// TwinCAT 3 PLC project Untitled1
// ProgramVersion: 3.1.4024.0
// libraries:
//   Tc2_EtherCAT, * (Beckhoff Automation GmbH)
//   Tc2_MC2, * (Beckhoff Automation GmbH)
//   Tc2_ModbusSrv, * (Beckhoff Automation GmbH)
//   Tc2_Standard, * (Beckhoff Automation GmbH)
//   Tc2_SUPS, * (Beckhoff Automation GmbH)
//   Tc2_System, * (Beckhoff Automation GmbH)
//   Tc2_Utilities, * (Beckhoff Automation GmbH)
//   Tc3_Module, * (Beckhoff Automation GmbH)
//   Util, * (System)
//   VisuDialogs, * (System)
// project tree:
//   02DUTs/Ads/ AutostoreControlCommand.TcDUT (not stored), AutostoreStatus.TcDUT, BarcodeVerificationResult.TcDUT, ButtonStatus.TcDUT, DigitalInputStatus.TcDUT (not stored), DigitalOutputStatus.TcDUT (not stored), EStopStatus.TcDUT, E_SAFETYDOOR.TcDUT, E_SafetyStates.TcDUT, FB_Application.TcPOU, FB_Light_tower_module.TcPOU, FB_Safety_module.TcPOU, FB_ToteData.TcPOU, FB_Tote_Subsystem.TcPOU, MachineControlCommand.TcDUT, MachineStatus.TcDUT, OrderToteCommand.TcDUT, OrderToteErrorStatus.TcDUT, SafetyDoorStatus.TcDUT, SafetyStatus.TcDUT, StationMode.TcDUT, ST_IO_16.TcDUT (not stored), ST_LightTower.TcDUT, ToteStatus.TcDUT, ToteSubsystemWorkflowStatus.TcDUT
//   GVLs/ GVL.TcGVL, GVL_IOLink.TcGVL, G_HMI.TcGVL, G_IO.TcGVL
//   / EtherCAT_Task.TcTTO, GlobalTextList.TcGTLO, MianTask.TcTTO, VisualizationManager.TcVMO (not stored), VISU_TASK.TcTTO
//   Mian/ Event_add.TcPOU, Event_clear.TcPOU, MAIN.TcPOU
//   Mian/machine/axis/ AxisHMI_Ex.TcVIS (not stored), E_HomingSteps.TcDUT (not stored), FB_MotionAxis_MC.TcPOU, MC_HomeAxis.TcPOU (not stored), ST_MotionAxis_MC.TcDUT
//   Mian/machine/bufferr module/ Buffer_roller.TcDUT (not stored), E_RollerStates.TcDUT, FB_buffer.TcPOU, FB_roller.TcPOU, Inbound_roller.TcDUT
//   Mian/machine/ FB_DigitalInput.TcPOU (not stored), FB_GPWM.TcPOU (not stored), Roller.TcDUT, Valve.TcDUT (not stored)
//   Mian/machine/loading moudle/ E_LoadingStates.TcDUT, E_Transfer.TcDUT, FB_loading.TcPOU, Roller_x.TcDUT, Roller_y.TcDUT
//   Mian/machine/mcp/ FB_mcp.TcPOU, ST_control_pannel.TcDUT (not stored), ST_safetyDoor.TcDUT
//   Mian/machine/working moudle/Estates/ E_Condition.TcDUT, E_WorkingStates.TcDUT
//   Mian/machine/working moudle/ FB_working.TcPOU, Inbound.TcDUT, Outbound.TcDUT
//   Mian/statemachine/ E_SystemManager.TcDUT, Prepare_Date_Time.TcPOU, ST_EVENT.TcDUT (not stored)
//   VISUs/VISUs/ Menu.TcVIS, visu_buffer.TcVIS, visu_loading.TcVIS, visu_main.TcVIS, visu_operation.TcVIS, visu_working.TcVIS, v_io_buffer.TcVIS, v_alarm.TcVIS, v_io_loading.TcVIS, v_io_working.TcVIS
// real-time tasks:
//   TASK PlcTask: cycle T#10ms, priority 20, ADS port 350
//   TASK EtherCAT_Task: cycle T#2ms, priority 1, ADS port 351
//   TASK VISU_TASK: cycle T#200000us, priority 30, ADS port 352
// motion (NC):
//   TASK NC-Task 1 SAF: cycle T#4ms, priority 4, ADS port 501
//   TASK NC-Task 1 SVB: cycle T#10ms, priority 8, ADS port 511
//   AXIS buffer_stopper (id 1)
//     PositionAreaControl: Enable=false
//     OtherSettings: AllowMotionCmdToSlave=true
//     encoder EncType=19
//       EncPara: ScaleFactorNumerator=36, ScaleFactorDenominator=8388608, MaxCount=#xffffffff, ReferenceSystem=1
//         Inc: RefSoftSyncMask=#x00800000
//     drive DrvType=16
//       DrvPara: MaxCount=#xffffffff, DriveControlDWord=#x00020100
//         Analog: TorqueSetpointScale=10, ScaleFactorActTorque=0.1
//         TimeComp: TaskDelayCycles=1
//     controller CtrType=1
//       CtrPara: PriorControlFactor=1
//         PosDiffControl: Enable=false
//         Observer: BandWidth=20
//   AXIS lift_motor (id 3)
//     PositionAreaControl: Enable=false
//     OtherSettings: AllowMotionCmdToSlave=true
//     encoder EncType=19
//       EncPara: ScaleFactorNumerator=3.97364299e-07, MaxCount=#xffffffff, ReferenceSystem=1
//     drive DrvType=16
//       DrvPara: MaxCount=#xffffffff, DriveControlDWord=#x00020100
//         Analog: TorqueSetpointScale=10, ScaleFactorActTorque=0.1
//         TimeComp: TaskDelayCycles=1
//     controller CtrType=1
//       CtrPara: PriorControlFactor=1
//         PosDiffControl: Enable=false
//         Observer: BandWidth=20
//   AXIS working_lift_motor (id 4)
//     PositionAreaControl: Enable=false
//     OtherSettings: AllowMotionCmdToSlave=true
//     encoder EncType=19
//       EncPara: ScaleFactorNumerator=5.96046448e-07, Inverse=true, MaxCount=#xffffffff, ReferenceSystem=1
//     drive DrvType=16
//       DrvPara: Inverse=true, MaxCount=#xffffffff, DriveControlDWord=#x00020100
//         Analog: TorqueSetpointScale=10, ScaleFactorActTorque=0.1
//         TimeComp: TaskDelayCycles=1
//     controller CtrType=1
//       CtrPara: PriorControlFactor=1
//         PosDiffControl: Enable=false
//         Observer: BandWidth=20
//   AXIS working_open_bag (id 5)
//     General: UnitName=°
//     PositionAreaControl: Enable=false
//     OtherSettings: AllowMotionCmdToSlave=true
//     encoder EncType=1
//       EncPara: ScaleFactorNumerator=36, ScaleFactorDenominator=8388608, ReferenceSystem=1
//         Inc: RefSoftSyncMask=#x00800000
//     drive DrvType=5
//       Analog: TorqueSetpointScale=10, ScaleFactorActTorque=0.1
//       TimeComp: TaskDelayCycles=1
//     controller CtrType=1
//       CtrPara: PriorControlFactor=1
//         PosDiffControl: Enable=false
//         Observer: BandWidth=20
//   AXIS bag_open_vacuun_0 (id 2)
//     General: UnitName=°
//     PositionAreaControl: Enable=false
//     OtherSettings: AllowMotionCmdToSlave=true
//     encoder EncType=19
//       EncPara: ScaleFactorNumerator=90, ScaleFactorDenominator=8388608, MaxCount=#xffffffff, ReferenceSystem=1
//         Inc: RefSoftSyncMask=#x00800000
//     drive DrvType=16
//       DrvPara: MaxCount=#xffffffff, DriveControlDWord=#x00020100
//         Analog: TorqueSetpointScale=10, ScaleFactorActTorque=0.1
//         TimeComp: TaskDelayCycles=1
//     controller CtrType=1
//       CtrPara: PriorControlFactor=1
//         PosDiffControl: Enable=false
//         Observer: BandWidth=20
//   AXIS bag_open_vacuun_1 (id 8)
//     General: UnitName=°
//     PositionAreaControl: Enable=false
//     OtherSettings: AllowMotionCmdToSlave=true
//     encoder EncType=19
//       EncPara: ScaleFactorNumerator=90, ScaleFactorDenominator=8388608, MaxCount=#xffffffff, ReferenceSystem=1
//         Inc: RefSoftSyncMask=#x00800000
//     drive DrvType=16
//       DrvPara: MaxCount=#xffffffff, DriveControlDWord=#x00020100
//         Analog: TorqueSetpointScale=10, ScaleFactorActTorque=0.1
//         TimeComp: TaskDelayCycles=1
//     controller CtrType=1
//       CtrPara: PriorControlFactor=1
//         PosDiffControl: Enable=false
//         Observer: BandWidth=20
//   AXIS bag_open_0 (id 9)
//     General: UnitName=°
//     PositionAreaControl: Enable=false
//     OtherSettings: AllowMotionCmdToSlave=true
//     encoder EncType=19
//       EncPara: ScaleFactorNumerator=360, ScaleFactorDenominator=8388608, MaxCount=#xffffffff, ReferenceSystem=1
//         Inc: RefSoftSyncMask=#x00800000
//     drive DrvType=16
//       DrvPara: MaxCount=#xffffffff, DriveControlDWord=#x00020100
//         Analog: TorqueSetpointScale=10, ScaleFactorActTorque=0.1
//         TimeComp: TaskDelayCycles=1
//     controller CtrType=1
//       CtrPara: PriorControlFactor=1
//         PosDiffControl: Enable=false
//         Observer: BandWidth=20
//   AXIS bag_open_1 (id 7)
//     General: UnitName=°
//     PositionAreaControl: Enable=false
//     OtherSettings: AllowMotionCmdToSlave=true
//     encoder EncType=19
//       EncPara: ScaleFactorNumerator=360, ScaleFactorDenominator=8388608, MaxCount=#xffffffff, ReferenceSystem=1
//         Inc: RefSoftSyncMask=#x00800000
//     drive DrvType=16
//       DrvPara: MaxCount=#xffffffff, DriveControlDWord=#x00020100
//         Analog: TorqueSetpointScale=10, ScaleFactorActTorque=0.1
//         TimeComp: TaskDelayCycles=1
//     controller CtrType=1
//       CtrPara: PriorControlFactor=1
//         PosDiffControl: Enable=false
//         Observer: BandWidth=20
//   AXIS bag_open_2 (id 10)
//     General: UnitName=°
//     PositionAreaControl: Enable=false
//     OtherSettings: AllowMotionCmdToSlave=true
//     encoder EncType=19
//       EncPara: ScaleFactorNumerator=360, ScaleFactorDenominator=8388608, MaxCount=#xffffffff, ReferenceSystem=1
//         Inc: RefSoftSyncMask=#x00800000
//     drive DrvType=16
//       DrvPara: MaxCount=#xffffffff, DriveControlDWord=#x00020100
//         Analog: TorqueSetpointScale=10, ScaleFactorActTorque=0.1
//         TimeComp: TaskDelayCycles=1
//     controller CtrType=1
//       CtrPara: PriorControlFactor=1
//         PosDiffControl: Enable=false
//         Observer: BandWidth=20
//   AXIS bag_open_3 (id 6)
//     General: UnitName=°
//     PositionAreaControl: Enable=false
//     OtherSettings: AllowMotionCmdToSlave=true
//     encoder EncType=19
//       EncPara: ScaleFactorNumerator=360, ScaleFactorDenominator=8388608, MaxCount=#xffffffff, ReferenceSystem=1
//         Inc: RefSoftSyncMask=#x00800000
//     drive DrvType=16
//       DrvPara: MaxCount=#xffffffff, DriveControlDWord=#x00020100
//         Analog: TorqueSetpointScale=10, ScaleFactorActTorque=0.1
//         TimeComp: TaskDelayCycles=1
//     controller CtrType=1
//       CtrPara: PriorControlFactor=1
//         PosDiffControl: Enable=false
//         Observer: BandWidth=20
// I/O:
//   DEVICE Device 1 (EtherCAT), AmsNetId 192.168.11.159.2.1
//     Term 1 (EK1200) [EK1200-5000 EtherCAT Power supply (2A E-Bus)]
//       mcp_di0 [EL1809 16Ch. Dig. Input 24V, 3ms]
//       mcp_do0 [EL2809-0015 16Ch. Dig. Output 24V DC, 0.35A, not short-circuit proof]
//       Term 4 (EL6910) [EL6910, TwinSAFE PLC]
//       Term 5 (EL1904) [EL1904, 4 Ch. Safety Input 24V, TwinSAFE]
//         modules: Module 1 (FSOES)
//       Term 6 (EL2904) [EL2904, 4 Ch. Safety Output 24V, 0.5A, TwinSAFE]
//         modules: Module 1 (FSOES), Module 2 (DO)
//       Term 41 (EL3064) [EL3064 4Ch. Ana. Input 0-10V]
//       Term 42 (EL6631-0010) [EL6631-0010 PROFINET IO Device]
//       Term 7 (EL9011) [EL9011 End Terminal]
//   DEVICE Device 4 (EtherCAT), AmsNetId 192.168.11.159.5.1
//     Box 8 (CU1128) [CU1128 6x EtherCAT junction]
//       buffer_io [EK1100 EtherCAT Coupler (2A E-Bus)]
//         buffer_di1 [EL1809 16Ch. Dig. Input 24V, 3ms]
//         buffer_di2 [EL1809 16Ch. Dig. Input 24V, 3ms]
//         buffer_do1 [EL2809-0015 16Ch. Dig. Output 24V DC, 0.35A, not short-circuit proof]
//         buffer_do2 [EL2809-0015 16Ch. Dig. Output 24V DC, 0.35A, not short-circuit proof] (disabled)
//         Term 14 (EL1904) [EL1904, 4 Ch. Safety Input 24V, TwinSAFE]
//           modules: Module 1 (FSOES)
//         Term 15 (EL2904) [EL2904, 4 Ch. Safety Output 24V, 0.5A, TwinSAFE]
//           modules: Module 1 (FSOES), Module 2 (DO)
//         Term 31 (EL9011) [EL9011 End Terminal]
//       buffer_stopper [SV660_1Axis_00915]
//       loading_io [EK1100 EtherCAT Coupler (2A E-Bus)]
//         lift_di3 [EL1809 16Ch. Dig. Input 24V, 3ms]
//         lift_di4 [EL1809 16Ch. Dig. Input 24V, 3ms]
//         lift_do3 [EL2809-0015 16Ch. Dig. Output 24V DC, 0.35A, not short-circuit proof]
//         lift_do4 [EL2809-0015 16Ch. Dig. Output 24V DC, 0.35A, not short-circuit proof]
//         Term 23 (EL1904) [EL1904, 4 Ch. Safety Input 24V, TwinSAFE]
//           modules: Module 1 (FSOES)
//         Term 24 (EL1904) [EL1904, 4 Ch. Safety Input 24V, TwinSAFE]
//           modules: Module 1 (FSOES)
//         Term 25 (EL2904) [EL2904, 4 Ch. Safety Output 24V, 0.5A, TwinSAFE]
//           modules: Module 1 (FSOES), Module 2 (DO)
//         Term 32 (EL9011) [EL9011 End Terminal]
//       loading_motor [SV635_1Axis_03411]
//       working_module [CU1128 6x EtherCAT junction - Dev A]
//         working_io [EK1100 EtherCAT Coupler (2A E-Bus)]
//           working_di5 [EL1809 16Ch. Dig. Input 24V, 3ms]
//           working_di6 [EL1809 16Ch. Dig. Input 24V, 3ms]
//           working_do5 [EL2809-0015 16Ch. Dig. Output 24V DC, 0.35A, not short-circuit proof]
//           working_do6 [EL2809-0015 16Ch. Dig. Output 24V DC, 0.35A, not short-circuit proof]
//           Term 33 (EL1904) [EL1904, 4 Ch. Safety Input 24V, TwinSAFE]
//             modules: Module 1 (FSOES)
//           Term 34 (EL2904) [EL2904, 4 Ch. Safety Output 24V, 0.5A, TwinSAFE]
//             modules: Module 1 (FSOES), Module 2 (DO)
//           Term 33 (EL9011) [EL9011 End Terminal]
//         working_liftmotor [SV635_1Axis_03411]
//         woking_openbag [SV635_1Axis_03411]
//         bag_open_dio [EK1100 EtherCAT Coupler (2A E-Bus)]
//           di7 [EL1809 16Ch. Dig. Input 24V, 3ms]
//           di8 [EL1809 16Ch. Dig. Input 24V, 3ms]
//           do7 [EL2809-0015 16Ch. Dig. Output 24V DC, 0.35A, not short-circuit proof]
//           Term 71 (EL9011) [EL9011 End Terminal]
//         bag_vacuun [SV660ND_2Axis_V1.00]
//           modules: Module 1 (CSP/CSV), Module 2 (CSP/CSV)
//         bag_open_0_1 [SV660ND_2Axis_V1.00]
//           modules: Module 1 (CSP/CSV), Module 2 (CSP/CSV)
//         bag_open_2_3 [SV660ND_2Axis_V1.00]
//           modules: Module 1 (CSP/CSV), Module 2 (CSP/CSV)
//       Term 37 (CU1128-C) [CU1128 6x EtherCAT junction - Dev B]
// variable links:
//   Device 1 (EtherCAT) <-> Device 1 (EtherCAT)/Term 1 (EK1200)/Term 4 (EL6910)
//     Term 1 (EK1200)/Term 5 (EL1904)/Module 1 (FSOES)/RxPDO/FSOE <-> ConnectionInputs/Message_3 TxPDO
//     Term 1 (EK1200)/Term 5 (EL1904)/Module 1 (FSOES)/TxPDO/FSOE <-> ConnectionOutputs/Message_3 RxPDO
//   Device 1 (EtherCAT) <-> Device 1 (EtherCAT)/Term 1 (EK1200)/Term 6 (EL2904)
//     Term 1 (EK1200)/Term 4 (EL6910)/ConnectionInputs/Message_4 TxPDO <-> Module 1 (FSOES)/RxPDO/FSOE
//     Term 1 (EK1200)/Term 4 (EL6910)/ConnectionOutputs/Message_4 RxPDO <-> Module 1 (FSOES)/TxPDO/FSOE
//   Device 1 (EtherCAT) <-> Device 4 (EtherCAT)/Box 8 (CU1128)/buffer_io/Term 14 (EL1904)
//     Term 1 (EK1200)/Term 4 (EL6910)/ConnectionInputs/Message_5 TxPDO <-> Module 1 (FSOES)/RxPDO/FSOE
//     Term 1 (EK1200)/Term 4 (EL6910)/ConnectionOutputs/Message_5 RxPDO <-> Module 1 (FSOES)/TxPDO/FSOE
//   Device 1 (EtherCAT) <-> Device 4 (EtherCAT)/Box 8 (CU1128)/buffer_io/Term 15 (EL2904)
//     Term 1 (EK1200)/Term 4 (EL6910)/ConnectionInputs/Message_6 TxPDO <-> Module 1 (FSOES)/RxPDO/FSOE
//     Term 1 (EK1200)/Term 4 (EL6910)/ConnectionOutputs/Message_6 RxPDO <-> Module 1 (FSOES)/TxPDO/FSOE
//   Device 1 (EtherCAT) <-> Device 4 (EtherCAT)/Box 8 (CU1128)/loading_io/Term 23 (EL1904)
//     Term 1 (EK1200)/Term 4 (EL6910)/ConnectionOutputs/Message_7 RxPDO <-> Module 1 (FSOES)/TxPDO/FSOE
//   Device 1 (EtherCAT) <-> Device 4 (EtherCAT)/Box 8 (CU1128)/loading_io/Term 25 (EL2904)
//     Term 1 (EK1200)/Term 4 (EL6910)/ConnectionInputs/Message_9 TxPDO <-> Module 1 (FSOES)/RxPDO/FSOE
//     Term 1 (EK1200)/Term 4 (EL6910)/ConnectionOutputs/Message_9 RxPDO <-> Module 1 (FSOES)/TxPDO/FSOE
//   Device 1 (EtherCAT) <-> Device 4 (EtherCAT)/Box 8 (CU1128)/working_module/working_io/Term 33 (EL1904)
//     Term 1 (EK1200)/Term 4 (EL6910)/ConnectionInputs/Message_10 TxPDO <-> Module 1 (FSOES)/RxPDO/FSOE
//     Term 1 (EK1200)/Term 4 (EL6910)/ConnectionOutputs/Message_10 RxPDO <-> Module 1 (FSOES)/TxPDO/FSOE
//   Device 1 (EtherCAT) <-> Device 4 (EtherCAT)/Box 8 (CU1128)/working_module/working_io/Term 34 (EL2904)
//     Term 1 (EK1200)/Term 4 (EL6910)/ConnectionInputs/Message_11 TxPDO <-> Module 1 (FSOES)/RxPDO/FSOE
//     Term 1 (EK1200)/Term 4 (EL6910)/ConnectionOutputs/Message_11 RxPDO <-> Module 1 (FSOES)/TxPDO/FSOE
//   Device 4 (EtherCAT) <-> Device 1 (EtherCAT)/Term 1 (EK1200)/Term 4 (EL6910)
//     Box 8 (CU1128)/loading_io/Term 23 (EL1904)/Module 1 (FSOES)/RxPDO/FSOE <-> ConnectionInputs/Message_7 TxPDO
//     Box 8 (CU1128)/loading_io/Term 24 (EL1904)/Module 1 (FSOES)/RxPDO/FSOE <-> ConnectionInputs/Message_8 TxPDO
//     Box 8 (CU1128)/loading_io/Term 24 (EL1904)/Module 1 (FSOES)/TxPDO/FSOE <-> ConnectionOutputs/Message_8 RxPDO
//   NC-Task 1 SAF/Axes/bag_open_0 <-> Device 4 (EtherCAT)/Box 8 (CU1128)/working_module/bag_open_0_1
//     Drive/Inputs/In/nDataIn1 <-> Module 1 (CSP/CSV)/Inputs/Following error actual value
//     Drive/Inputs/In/nDcOutputTime <-> InfoData/DcOutputShift
//     Drive/Inputs/In/nState1 <-> Module 1 (CSP/CSV)/Inputs/StatusWord
//     Drive/Inputs/In/nState2 <-> Module 1 (CSP/CSV)/Inputs/StatusWord @bit 8
//     Drive/Inputs/In/nState4 @bit 1 <-> WcState/InputToggle
//     Drive/Inputs/In/nState4 <-> WcState/WcState
//     Drive/Inputs/In/nState5 <-> Module 1 (CSP/CSV)/Inputs/Modes of Operation Display
//     Drive/Outputs/Out/nCtrl1 <-> Module 1 (CSP/CSV)/Outputs/ControlWord
//     Drive/Outputs/Out/nCtrl2 <-> Module 1 (CSP/CSV)/Outputs/ControlWord @bit 8
//     Drive/Outputs/Out/nCtrl5 <-> Module 1 (CSP/CSV)/Outputs/Modes of Operation
//     Drive/Outputs/Out/nDataOut1 <-> Module 1 (CSP/CSV)/Outputs/Target position
//     Drive/Outputs/Out/nDataOut2 <-> Module 1 (CSP/CSV)/Outputs/Target velocity
//     Enc/Inputs/In/nDataIn1 <-> Module 1 (CSP/CSV)/Inputs/Position actual value
//     Enc/Inputs/In/nDataIn3 <-> Module 1 (CSP/CSV)/Inputs/Touch probe pos1 pos value
//     Enc/Inputs/In/nDataIn5 <-> Module 1 (CSP/CSV)/Inputs/Touch probe pos2 pos value
//     Enc/Inputs/In/nDataIn7 <-> Module 1 (CSP/CSV)/Inputs/ActualVelocity
//     Enc/Inputs/In/nDcInputTime <-> InfoData/DcInputShift
//     Enc/Inputs/In/nState4 @bit 1 <-> WcState/InputToggle
//     Enc/Inputs/In/nState4 <-> WcState/WcState
//     Enc/Inputs/In/nState5 <-> Module 1 (CSP/CSV)/Inputs/Touch probe status
//     Enc/Inputs/In/nState6 <-> Module 1 (CSP/CSV)/Inputs/Touch probe status @bit 8
//     Enc/Outputs/Out/nCtrl5 <-> Module 1 (CSP/CSV)/Outputs/Touch probe function
//     Enc/Outputs/Out/nCtrl6 <-> Module 1 (CSP/CSV)/Outputs/Touch probe function @bit 8
//   NC-Task 1 SAF/Axes/bag_open_1 <-> Device 4 (EtherCAT)/Box 8 (CU1128)/working_module/bag_open_0_1
//     Drive/Inputs/In/nDataIn1 <-> Module 2 (CSP/CSV)/Inputs/Following error actual value
//     Drive/Inputs/In/nDcOutputTime <-> InfoData/DcOutputShift
//     Drive/Inputs/In/nState1 <-> Module 2 (CSP/CSV)/Inputs/StatusWord
//     Drive/Inputs/In/nState2 <-> Module 2 (CSP/CSV)/Inputs/StatusWord @bit 8
//     Drive/Inputs/In/nState4 @bit 1 <-> WcState/InputToggle
//     Drive/Inputs/In/nState4 <-> WcState/WcState
//     Drive/Inputs/In/nState5 <-> Module 2 (CSP/CSV)/Inputs/Modes of Operation Display
//     Drive/Outputs/Out/nCtrl1 <-> Module 2 (CSP/CSV)/Outputs/ControlWord
//     Drive/Outputs/Out/nCtrl2 <-> Module 2 (CSP/CSV)/Outputs/ControlWord @bit 8
//     Drive/Outputs/Out/nCtrl5 <-> Module 2 (CSP/CSV)/Outputs/Modes of Operation
//     Drive/Outputs/Out/nDataOut1 <-> Module 2 (CSP/CSV)/Outputs/Target position
//     Drive/Outputs/Out/nDataOut2 <-> Module 2 (CSP/CSV)/Outputs/Target velocity
//     Enc/Inputs/In/nDataIn1 <-> Module 2 (CSP/CSV)/Inputs/Position actual value
//     Enc/Inputs/In/nDataIn3 <-> Module 2 (CSP/CSV)/Inputs/Touch probe pos1 pos value
//     Enc/Inputs/In/nDataIn5 <-> Module 2 (CSP/CSV)/Inputs/Touch probe pos2 pos value
//     Enc/Inputs/In/nDataIn7 <-> Module 2 (CSP/CSV)/Inputs/ActualVelocity
//     Enc/Inputs/In/nDcInputTime <-> InfoData/DcInputShift
//     Enc/Inputs/In/nState4 @bit 1 <-> WcState/InputToggle
//     Enc/Inputs/In/nState4 <-> WcState/WcState
//     Enc/Inputs/In/nState5 <-> Module 2 (CSP/CSV)/Inputs/Touch probe status
//     Enc/Inputs/In/nState6 <-> Module 2 (CSP/CSV)/Inputs/Touch probe status @bit 8
//     Enc/Outputs/Out/nCtrl5 <-> Module 2 (CSP/CSV)/Outputs/Touch probe function
//     Enc/Outputs/Out/nCtrl6 <-> Module 2 (CSP/CSV)/Outputs/Touch probe function @bit 8
//   NC-Task 1 SAF/Axes/bag_open_2 <-> Device 4 (EtherCAT)/Box 8 (CU1128)/working_module/bag_open_2_3
//     Drive/Inputs/In/nDataIn1 <-> Module 1 (CSP/CSV)/Inputs/Following error actual value
//     Drive/Inputs/In/nDcOutputTime <-> InfoData/DcOutputShift
//     Drive/Inputs/In/nState1 <-> Module 1 (CSP/CSV)/Inputs/StatusWord
//     Drive/Inputs/In/nState2 <-> Module 1 (CSP/CSV)/Inputs/StatusWord @bit 8
//     Drive/Inputs/In/nState4 @bit 1 <-> WcState/InputToggle
//     Drive/Inputs/In/nState4 <-> WcState/WcState
//     Drive/Inputs/In/nState5 <-> Module 1 (CSP/CSV)/Inputs/Modes of Operation Display
//     Drive/Outputs/Out/nCtrl1 <-> Module 1 (CSP/CSV)/Outputs/ControlWord
//     Drive/Outputs/Out/nCtrl2 <-> Module 1 (CSP/CSV)/Outputs/ControlWord @bit 8
//     Drive/Outputs/Out/nCtrl5 <-> Module 1 (CSP/CSV)/Outputs/Modes of Operation
//     Drive/Outputs/Out/nDataOut1 <-> Module 1 (CSP/CSV)/Outputs/Target position
//     Drive/Outputs/Out/nDataOut2 <-> Module 1 (CSP/CSV)/Outputs/Target velocity
//     Enc/Inputs/In/nDataIn1 <-> Module 1 (CSP/CSV)/Inputs/Position actual value
//     Enc/Inputs/In/nDataIn3 <-> Module 1 (CSP/CSV)/Inputs/Touch probe pos1 pos value
//     Enc/Inputs/In/nDataIn5 <-> Module 1 (CSP/CSV)/Inputs/Touch probe pos2 pos value
//     Enc/Inputs/In/nDataIn7 <-> Module 1 (CSP/CSV)/Inputs/ActualVelocity
//     Enc/Inputs/In/nDcInputTime <-> InfoData/DcInputShift
//     Enc/Inputs/In/nState4 @bit 1 <-> WcState/InputToggle
//     Enc/Inputs/In/nState4 <-> WcState/WcState
//     Enc/Inputs/In/nState5 <-> Module 1 (CSP/CSV)/Inputs/Touch probe status
//     Enc/Inputs/In/nState6 <-> Module 1 (CSP/CSV)/Inputs/Touch probe status @bit 8
//     Enc/Outputs/Out/nCtrl5 <-> Module 1 (CSP/CSV)/Outputs/Touch probe function
//     Enc/Outputs/Out/nCtrl6 <-> Module 1 (CSP/CSV)/Outputs/Touch probe function @bit 8
//   NC-Task 1 SAF/Axes/bag_open_3 <-> Device 4 (EtherCAT)/Box 8 (CU1128)/working_module/bag_open_2_3
//     Drive/Inputs/In/nDataIn1 <-> Module 2 (CSP/CSV)/Inputs/Following error actual value
//     Drive/Inputs/In/nDcOutputTime <-> InfoData/DcOutputShift
//     Drive/Inputs/In/nState1 <-> Module 2 (CSP/CSV)/Inputs/StatusWord
//     Drive/Inputs/In/nState2 <-> Module 2 (CSP/CSV)/Inputs/StatusWord @bit 8
//     Drive/Inputs/In/nState4 @bit 1 <-> WcState/InputToggle
//     Drive/Inputs/In/nState4 <-> WcState/WcState
//     Drive/Inputs/In/nState5 <-> Module 2 (CSP/CSV)/Inputs/Modes of Operation Display
//     Drive/Outputs/Out/nCtrl1 <-> Module 2 (CSP/CSV)/Outputs/ControlWord
//     Drive/Outputs/Out/nCtrl2 <-> Module 2 (CSP/CSV)/Outputs/ControlWord @bit 8
//     Drive/Outputs/Out/nCtrl5 <-> Module 2 (CSP/CSV)/Outputs/Modes of Operation
//     Drive/Outputs/Out/nDataOut1 <-> Module 2 (CSP/CSV)/Outputs/Target position
//     Drive/Outputs/Out/nDataOut2 <-> Module 2 (CSP/CSV)/Outputs/Target velocity
//     Enc/Inputs/In/nDataIn1 <-> Module 2 (CSP/CSV)/Inputs/Position actual value
//     Enc/Inputs/In/nDataIn3 <-> Module 2 (CSP/CSV)/Inputs/Touch probe pos1 pos value
//     Enc/Inputs/In/nDataIn5 <-> Module 2 (CSP/CSV)/Inputs/Touch probe pos2 pos value
//     Enc/Inputs/In/nDataIn7 <-> Module 2 (CSP/CSV)/Inputs/ActualVelocity
//     Enc/Inputs/In/nDcInputTime <-> InfoData/DcInputShift
//     Enc/Inputs/In/nState4 @bit 1 <-> WcState/InputToggle
//     Enc/Inputs/In/nState4 <-> WcState/WcState
//     Enc/Inputs/In/nState5 <-> Module 2 (CSP/CSV)/Inputs/Touch probe status
//     Enc/Inputs/In/nState6 <-> Module 2 (CSP/CSV)/Inputs/Touch probe status @bit 8
//     Enc/Outputs/Out/nCtrl5 <-> Module 2 (CSP/CSV)/Outputs/Touch probe function
//     Enc/Outputs/Out/nCtrl6 <-> Module 2 (CSP/CSV)/Outputs/Touch probe function @bit 8
//   NC-Task 1 SAF/Axes/bag_open_vacuun_0 <-> Device 4 (EtherCAT)/Box 8 (CU1128)/working_module/bag_vacuun
//     Drive/Inputs/In/nDataIn1 <-> Module 1 (CSP/CSV)/Inputs/Following error actual value
//     Drive/Inputs/In/nDcOutputTime <-> InfoData/DcOutputShift
//     Drive/Inputs/In/nState1 <-> Module 1 (CSP/CSV)/Inputs/StatusWord
//     Drive/Inputs/In/nState2 <-> Module 1 (CSP/CSV)/Inputs/StatusWord @bit 8
//     Drive/Inputs/In/nState4 @bit 1 <-> WcState/InputToggle
//     Drive/Inputs/In/nState4 <-> WcState/WcState
//     Drive/Inputs/In/nState5 <-> Module 1 (CSP/CSV)/Inputs/Modes of Operation Display
//     Drive/Outputs/Out/nCtrl1 <-> Module 1 (CSP/CSV)/Outputs/ControlWord
//     Drive/Outputs/Out/nCtrl2 <-> Module 1 (CSP/CSV)/Outputs/ControlWord @bit 8
//     Drive/Outputs/Out/nCtrl5 <-> Module 1 (CSP/CSV)/Outputs/Modes of Operation
//     Drive/Outputs/Out/nDataOut1 <-> Module 1 (CSP/CSV)/Outputs/Target position
//     Drive/Outputs/Out/nDataOut2 <-> Module 1 (CSP/CSV)/Outputs/Target velocity
//     Enc/Inputs/In/nDataIn1 <-> Module 1 (CSP/CSV)/Inputs/Position actual value
//     Enc/Inputs/In/nDataIn3 <-> Module 1 (CSP/CSV)/Inputs/Touch probe pos1 pos value
//     Enc/Inputs/In/nDataIn5 <-> Module 1 (CSP/CSV)/Inputs/Touch probe pos2 pos value
//     Enc/Inputs/In/nDataIn7 <-> Module 1 (CSP/CSV)/Inputs/ActualVelocity
//     Enc/Inputs/In/nDcInputTime <-> InfoData/DcInputShift
//     Enc/Inputs/In/nState4 @bit 1 <-> WcState/InputToggle
//     Enc/Inputs/In/nState4 <-> WcState/WcState
//     Enc/Inputs/In/nState5 <-> Module 1 (CSP/CSV)/Inputs/Touch probe status
//     Enc/Inputs/In/nState6 <-> Module 1 (CSP/CSV)/Inputs/Touch probe status @bit 8
//     Enc/Outputs/Out/nCtrl5 <-> Module 1 (CSP/CSV)/Outputs/Touch probe function
//     Enc/Outputs/Out/nCtrl6 <-> Module 1 (CSP/CSV)/Outputs/Touch probe function @bit 8
//   NC-Task 1 SAF/Axes/bag_open_vacuun_1 <-> Device 4 (EtherCAT)/Box 8 (CU1128)/working_module/bag_vacuun
//     Drive/Inputs/In/nDataIn1 <-> Module 2 (CSP/CSV)/Inputs/Following error actual value
//     Drive/Inputs/In/nDcOutputTime <-> InfoData/DcOutputShift
//     Drive/Inputs/In/nState1 <-> Module 2 (CSP/CSV)/Inputs/StatusWord
//     Drive/Inputs/In/nState2 <-> Module 2 (CSP/CSV)/Inputs/StatusWord @bit 8
//     Drive/Inputs/In/nState4 @bit 1 <-> WcState/InputToggle
//     Drive/Inputs/In/nState4 <-> WcState/WcState
//     Drive/Inputs/In/nState5 <-> Module 2 (CSP/CSV)/Inputs/Modes of Operation Display
//     Drive/Outputs/Out/nCtrl1 <-> Module 2 (CSP/CSV)/Outputs/ControlWord
//     Drive/Outputs/Out/nCtrl2 <-> Module 2 (CSP/CSV)/Outputs/ControlWord @bit 8
//     Drive/Outputs/Out/nCtrl5 <-> Module 2 (CSP/CSV)/Outputs/Modes of Operation
//     Drive/Outputs/Out/nDataOut1 <-> Module 2 (CSP/CSV)/Outputs/Target position
//     Drive/Outputs/Out/nDataOut2 <-> Module 2 (CSP/CSV)/Outputs/Target velocity
//     Enc/Inputs/In/nDataIn1 <-> Module 2 (CSP/CSV)/Inputs/Position actual value
//     Enc/Inputs/In/nDataIn3 <-> Module 2 (CSP/CSV)/Inputs/Touch probe pos1 pos value
//     Enc/Inputs/In/nDataIn5 <-> Module 2 (CSP/CSV)/Inputs/Touch probe pos2 pos value
//     Enc/Inputs/In/nDataIn7 <-> Module 2 (CSP/CSV)/Inputs/ActualVelocity
//     Enc/Inputs/In/nDcInputTime <-> InfoData/DcInputShift
//     Enc/Inputs/In/nState4 @bit 1 <-> WcState/InputToggle
//     Enc/Inputs/In/nState4 <-> WcState/WcState
//     Enc/Inputs/In/nState5 <-> Module 2 (CSP/CSV)/Inputs/Touch probe status
//     Enc/Inputs/In/nState6 <-> Module 2 (CSP/CSV)/Inputs/Touch probe status @bit 8
//     Enc/Outputs/Out/nCtrl5 <-> Module 2 (CSP/CSV)/Outputs/Touch probe function
//     Enc/Outputs/Out/nCtrl6 <-> Module 2 (CSP/CSV)/Outputs/Touch probe function @bit 8
//   NC-Task 1 SAF/Axes/buffer_stopper <-> Device 4 (EtherCAT)/Box 8 (CU1128)/buffer_stopper
//     Drive/Inputs/In/nDataIn1 <-> Inputs/Following error actual value
//     Drive/Inputs/In/nDataIn3[0] <-> Inputs/Torque actual value
//     Drive/Inputs/In/nDcOutputTime <-> InfoData/DcOutputShift
//     Drive/Inputs/In/nState1 <-> Inputs/Statusword
//     Drive/Inputs/In/nState2 <-> Inputs/Statusword @bit 8
//     Drive/Inputs/In/nState4 @bit 1 <-> WcState/InputToggle
//     Drive/Inputs/In/nState4 <-> WcState/WcState
//     Drive/Outputs/Out/nCtrl1 <-> Outputs/Controlword
//     Drive/Outputs/Out/nCtrl2 <-> Outputs/Controlword @bit 8
//     Drive/Outputs/Out/nDataOut1 <-> Outputs/Target position
//     Enc/Inputs/In/nDataIn1 <-> Inputs/Position actual value
//     Enc/Inputs/In/nDataIn3 <-> Inputs/Touch probe pos1 pos value
//     Enc/Inputs/In/nDataIn5 <-> Inputs/Touch probe pos2 pos value
//     Enc/Inputs/In/nDcInputTime <-> InfoData/DcInputShift
//     Enc/Inputs/In/nState4 @bit 1 <-> WcState/InputToggle
//     Enc/Inputs/In/nState4 <-> WcState/WcState
//     Enc/Inputs/In/nState5 <-> Inputs/Touch probe status
//     Enc/Inputs/In/nState6 <-> Inputs/Touch probe status @bit 8
//     Enc/Outputs/Out/nCtrl5 <-> Outputs/Touch probe function
//     Enc/Outputs/Out/nCtrl6 <-> Outputs/Touch probe function @bit 8
//   NC-Task 1 SAF/Axes/lift_motor <-> Device 4 (EtherCAT)/Box 8 (CU1128)/loading_motor
//     Drive/Inputs/In/nDataIn1 <-> Inputs/Following error actual value
//     Drive/Inputs/In/nDataIn3[0] <-> Inputs/Torque actual value
//     Drive/Inputs/In/nDcOutputTime <-> InfoData/DcOutputShift
//     Drive/Inputs/In/nState1 <-> Inputs/Statusword
//     Drive/Inputs/In/nState2 <-> Inputs/Statusword @bit 8
//     Drive/Inputs/In/nState4 @bit 1 <-> WcState/InputToggle
//     Drive/Inputs/In/nState4 <-> WcState/WcState
//     Drive/Outputs/Out/nCtrl1 <-> Outputs/Controlword
//     Drive/Outputs/Out/nCtrl2 <-> Outputs/Controlword @bit 8
//     Drive/Outputs/Out/nDataOut1 <-> Outputs/Target position
//     Enc/Inputs/In/nDataIn1 <-> Inputs/Position actual value
//     Enc/Inputs/In/nDataIn3 <-> Inputs/Touch probe pos1 pos value
//     Enc/Inputs/In/nDataIn5 <-> Inputs/Touch probe pos2 pos value
//     Enc/Inputs/In/nDcInputTime <-> InfoData/DcInputShift
//     Enc/Inputs/In/nState4 @bit 1 <-> WcState/InputToggle
//     Enc/Inputs/In/nState4 <-> WcState/WcState
//     Enc/Inputs/In/nState5 <-> Inputs/Touch probe status
//     Enc/Inputs/In/nState6 <-> Inputs/Touch probe status @bit 8
//     Enc/Outputs/Out/nCtrl5 <-> Outputs/Touch probe function
//     Enc/Outputs/Out/nCtrl6 <-> Outputs/Touch probe function @bit 8
//   NC-Task 1 SAF/Axes/working_lift_motor <-> Device 4 (EtherCAT)/Box 8 (CU1128)/working_module/working_liftmotor
//     Drive/Inputs/In/nDataIn1 <-> Inputs/Following error actual value
//     Drive/Inputs/In/nDataIn3[0] <-> Inputs/Torque actual value
//     Drive/Inputs/In/nDcOutputTime <-> InfoData/DcOutputShift
//     Drive/Inputs/In/nState1 <-> Inputs/Statusword
//     Drive/Inputs/In/nState2 <-> Inputs/Statusword @bit 8
//     Drive/Inputs/In/nState4 @bit 1 <-> WcState/InputToggle
//     Drive/Inputs/In/nState4 <-> WcState/WcState
//     Drive/Outputs/Out/nCtrl1 <-> Outputs/Controlword
//     Drive/Outputs/Out/nCtrl2 <-> Outputs/Controlword @bit 8
//     Drive/Outputs/Out/nDataOut1 <-> Outputs/Target position
//     Enc/Inputs/In/nDataIn1 <-> Inputs/Position actual value
//     Enc/Inputs/In/nDataIn3 <-> Inputs/Touch probe pos1 pos value
//     Enc/Inputs/In/nDataIn5 <-> Inputs/Touch probe pos2 pos value
//     Enc/Inputs/In/nDcInputTime <-> InfoData/DcInputShift
//     Enc/Inputs/In/nState4 @bit 1 <-> WcState/InputToggle
//     Enc/Inputs/In/nState4 <-> WcState/WcState
//     Enc/Inputs/In/nState5 <-> Inputs/Touch probe status
//     Enc/Inputs/In/nState6 <-> Inputs/Touch probe status @bit 8
//     Enc/Outputs/Out/nCtrl5 <-> Outputs/Touch probe function
//     Enc/Outputs/Out/nCtrl6 <-> Outputs/Touch probe function @bit 8
//   Untitled1/Untitled1 Instance <-> Device 1 (EtherCAT)/Term 1 (EK1200)/Term 4 (EL6910)
//     MianTask Inputs/GVL_IOLink.SO0_0 <-> StandardInputs/Standard Out Var 22
//     MianTask Inputs/GVL_IOLink.SO0_1 <-> StandardInputs/Standard Out Var 21
//     MianTask Inputs/GVL_IOLink.SO1_0 <-> StandardInputs/Standard Out Var 25
//     MianTask Inputs/GVL_IOLink.SO2_0 <-> StandardInputs/Standard Out Var 23
//     MianTask Inputs/GVL_IOLink.SO3_0 <-> StandardInputs/Standard Out Var 24
//     MianTask Inputs/GVL_IOLink.b_CoMerror <-> StandardInputs/Standard Out Var 15
//     MianTask Inputs/GVL_IOLink.b_FBerror <-> StandardInputs/Standard Out Var 14
//     MianTask Outputs/GVL_IOLink.PickModule_STO_EDM <-> StandardOutputs/Standard In Var 30
//     MianTask Outputs/GVL_IOLink.Rolller_belt_STO_EDM <-> StandardOutputs/Standard In Var 29
//     MianTask Outputs/GVL_IOLink.SPtop_EDM <-> StandardOutputs/Standard In Var 31
//     MianTask Outputs/GVL_IOLink.bMultingEnable <-> StandardOutputs/Standard In Var 26
//     MianTask Outputs/GVL_IOLink.bShield_light_curtain_Left <-> StandardOutputs/Standard In Var 16
//     MianTask Outputs/GVL_IOLink.bShield_light_curtain_Right <-> StandardOutputs/Standard In Var 17
//     MianTask Outputs/GVL_IOLink.b_EStopRestart <-> StandardOutputs/Standard In Var 13
//     MianTask Outputs/GVL_IOLink.b_ErrorAck <-> StandardOutputs/Standard In Var 1
//     MianTask Outputs/GVL_IOLink.b_GroupRun <-> StandardOutputs/Standard In Var 2
//     MianTask Outputs/GVL_IOLink.light_STO_EDM <-> StandardOutputs/Standard In Var 27
//     MianTask Outputs/GVL_IOLink.robot_eas_edm <-> StandardOutputs/Standard In Var 28
//   Untitled1/Untitled1 Instance <-> Device 1 (EtherCAT)/Term 1 (EK1200)/Term 5 (EL1904)
//     MianTask Inputs/GVL_IOLink.SI0_{0..3} <-> Module 1 (FSOES)/TxPDO/FSOE/InputChannel{1..4}  (4 links)
//   Untitled1/Untitled1 Instance <-> Device 1 (EtherCAT)/Term 1 (EK1200)/mcp_di0
//     MianTask Inputs/G_IO.arDI[0]/Ch[{0..15}] <-> Channel {1..16}/Input  (16 links)
//   Untitled1/Untitled1 Instance <-> Device 1 (EtherCAT)/Term 1 (EK1200)/mcp_do0
//     MianTask Outputs/G_IO.arDO[0]/Ch[{0..15}] <-> Channel {1..16}/Output  (16 links)
//   Untitled1/Untitled1 Instance <-> Device 4 (EtherCAT)/Box 8 (CU1128)/buffer_io/Term 14 (EL1904)
//     MianTask Inputs/GVL_IOLink.SI1_{0..3} <-> Module 1 (FSOES)/TxPDO/FSOE/InputChannel{1..4}  (4 links)
//   Untitled1/Untitled1 Instance <-> Device 4 (EtherCAT)/Box 8 (CU1128)/buffer_io/buffer_di1
//     MianTask Inputs/G_IO.arDI[1]/Ch[{0..15}] <-> Channel {1..16}/Input  (16 links)
//   Untitled1/Untitled1 Instance <-> Device 4 (EtherCAT)/Box 8 (CU1128)/buffer_io/buffer_di2
//     MianTask Inputs/G_IO.arDI[2]/Ch[{0..15}] <-> Channel {1..16}/Input  (16 links)
//   Untitled1/Untitled1 Instance <-> Device 4 (EtherCAT)/Box 8 (CU1128)/buffer_io/buffer_do1
//     MianTask Outputs/G_IO.arDO[1]/Ch[{0..15}] <-> Channel {1..16}/Output  (16 links)
//   Untitled1/Untitled1 Instance <-> Device 4 (EtherCAT)/Box 8 (CU1128)/buffer_io/buffer_do2
//     MianTask Outputs/G_IO.arDO[2]/Ch[{0..15}] <-> Channel {1..16}/Output  (16 links)
//   Untitled1/Untitled1 Instance <-> Device 4 (EtherCAT)/Box 8 (CU1128)/loading_io/Term 23 (EL1904)
//     MianTask Inputs/GVL_IOLink.SI2_{0..3} <-> Module 1 (FSOES)/TxPDO/FSOE/InputChannel{1..4}  (4 links)
//   Untitled1/Untitled1 Instance <-> Device 4 (EtherCAT)/Box 8 (CU1128)/loading_io/Term 24 (EL1904)
//     MianTask Inputs/GVL_IOLink.SI3_{0..3} <-> Module 1 (FSOES)/TxPDO/FSOE/InputChannel{1..4}  (4 links)
//   Untitled1/Untitled1 Instance <-> Device 4 (EtherCAT)/Box 8 (CU1128)/loading_io/lift_di3
//     MianTask Inputs/G_IO.arDI[3]/Ch[{0..15}] <-> Channel {1..16}/Input  (16 links)
//   Untitled1/Untitled1 Instance <-> Device 4 (EtherCAT)/Box 8 (CU1128)/loading_io/lift_di4
//     MianTask Inputs/G_IO.arDI[4]/Ch[{0..15}] <-> Channel {1..16}/Input  (16 links)
//   Untitled1/Untitled1 Instance <-> Device 4 (EtherCAT)/Box 8 (CU1128)/loading_io/lift_do3
//     MianTask Outputs/G_IO.arDO[3]/Ch[{0..15}] <-> Channel {1..16}/Output  (16 links)
//   Untitled1/Untitled1 Instance <-> Device 4 (EtherCAT)/Box 8 (CU1128)/loading_io/lift_do4
//     MianTask Outputs/G_IO.arDO[4]/Ch[{0..15}] <-> Channel {1..16}/Output  (16 links)
//   Untitled1/Untitled1 Instance <-> Device 4 (EtherCAT)/Box 8 (CU1128)/working_module/bag_open_dio/di7
//     MianTask Inputs/G_IO.arDI[7]/Ch[{0..15}] <-> Channel {1..16}/Input  (16 links)
//   Untitled1/Untitled1 Instance <-> Device 4 (EtherCAT)/Box 8 (CU1128)/working_module/bag_open_dio/di8
//     MianTask Inputs/G_IO.arDI[8]/Ch[{0..15}] <-> Channel {1..16}/Input  (16 links)
//   Untitled1/Untitled1 Instance <-> Device 4 (EtherCAT)/Box 8 (CU1128)/working_module/bag_open_dio/do7
//     MianTask Outputs/G_IO.arDO[7]/Ch[{0..15}] <-> Channel {1..16}/Output  (16 links)
//   Untitled1/Untitled1 Instance <-> Device 4 (EtherCAT)/Box 8 (CU1128)/working_module/working_io/working_di5
//     MianTask Inputs/G_IO.arDI[5]/Ch[{0..15}] <-> Channel {1..16}/Input  (16 links)
//   Untitled1/Untitled1 Instance <-> Device 4 (EtherCAT)/Box 8 (CU1128)/working_module/working_io/working_di6
//     MianTask Inputs/G_IO.arDI[6]/Ch[{0..15}] <-> Channel {1..16}/Input  (16 links)
//   Untitled1/Untitled1 Instance <-> Device 4 (EtherCAT)/Box 8 (CU1128)/working_module/working_io/working_do5
//     MianTask Outputs/G_IO.arDO[5]/Ch[{0..15}] <-> Channel {1..16}/Output  (16 links)
//   Untitled1/Untitled1 Instance <-> Device 4 (EtherCAT)/Box 8 (CU1128)/working_module/working_io/working_do6
//     MianTask Outputs/G_IO.arDO[6]/Ch[{0..15}] <-> Channel {1..16}/Output  (16 links)
//   Untitled1/Untitled1 Instance <-> NC-Task 1 SAF/Axes/bag_open_0
//     MianTask Inputs/GVL.fb_working.AxisRef_bagOpen[0].NcToPlc <-> Outputs/ToPlc
//     MianTask Outputs/GVL.fb_working.AxisRef_bagOpen[0].PlcToNc <-> Inputs/FromPlc
//   Untitled1/Untitled1 Instance <-> NC-Task 1 SAF/Axes/bag_open_1
//     MianTask Inputs/GVL.fb_working.AxisRef_bagOpen[1].NcToPlc <-> Outputs/ToPlc
//     MianTask Outputs/GVL.fb_working.AxisRef_bagOpen[1].PlcToNc <-> Inputs/FromPlc
//   Untitled1/Untitled1 Instance <-> NC-Task 1 SAF/Axes/bag_open_2
//     MianTask Inputs/GVL.fb_working.AxisRef_bagOpen[2].NcToPlc <-> Outputs/ToPlc
//     MianTask Outputs/GVL.fb_working.AxisRef_bagOpen[2].PlcToNc <-> Inputs/FromPlc
//   Untitled1/Untitled1 Instance <-> NC-Task 1 SAF/Axes/bag_open_3
//     MianTask Inputs/GVL.fb_working.AxisRef_bagOpen[3].NcToPlc <-> Outputs/ToPlc
//     MianTask Outputs/GVL.fb_working.AxisRef_bagOpen[3].PlcToNc <-> Inputs/FromPlc
//   Untitled1/Untitled1 Instance <-> NC-Task 1 SAF/Axes/bag_open_vacuun_0
//     MianTask Inputs/GVL.fb_working.AxisRef_vacuun[0].NcToPlc <-> Outputs/ToPlc
//     MianTask Outputs/GVL.fb_working.AxisRef_vacuun[0].PlcToNc <-> Inputs/FromPlc
//   Untitled1/Untitled1 Instance <-> NC-Task 1 SAF/Axes/bag_open_vacuun_1
//     MianTask Inputs/GVL.fb_working.AxisRef_vacuun[1].NcToPlc <-> Outputs/ToPlc
//     MianTask Outputs/GVL.fb_working.AxisRef_vacuun[1].PlcToNc <-> Inputs/FromPlc
//   Untitled1/Untitled1 Instance <-> NC-Task 1 SAF/Axes/buffer_stopper
//     MianTask Inputs/GVL.fb_buffer.fb_rollers[3].AxisRef.NcToPlc <-> Outputs/ToPlc
//     MianTask Outputs/GVL.fb_buffer.fb_rollers[3].AxisRef.PlcToNc <-> Inputs/FromPlc
//   Untitled1/Untitled1 Instance <-> NC-Task 1 SAF/Axes/lift_motor
//     MianTask Inputs/GVL.fb_loading.AxisRef.NcToPlc <-> Outputs/ToPlc
//     MianTask Outputs/GVL.fb_loading.AxisRef.PlcToNc <-> Inputs/FromPlc
//   Untitled1/Untitled1 Instance <-> NC-Task 1 SAF/Axes/working_lift_motor
//     MianTask Inputs/GVL.fb_working.AxisRef_lift.NcToPlc <-> Outputs/ToPlc
//     MianTask Outputs/GVL.fb_working.AxisRef_lift.PlcToNc <-> Inputs/FromPlc
//   Untitled1/Untitled1 Instance <-> NC-Task 1 SAF/Axes/working_open_bag
//     MianTask Inputs/GVL.fb_working.AxisRef_bag.NcToPlc <-> Outputs/ToPlc
//     MianTask Outputs/GVL.fb_working.AxisRef_bag.PlcToNc <-> Inputs/FromPlc

CONFIGURATION Untitled1
    RESOURCE PLC ON TwinCAT3
        TASK EtherCAT_Task(INTERVAL := T#2ms, PRIORITY := 1);
        TASK MianTask(INTERVAL := T#10ms, PRIORITY := 20);
        TASK VISU_TASK(INTERVAL := T#200000us, PRIORITY := 30);
        PROGRAM MAIN WITH MianTask : MAIN;
        PROGRAM VisuElems_Visu_Prg WITH VISU_TASK : VisuElems.Visu_Prg;
    END_RESOURCE
END_CONFIGURATION

// ---- 02DUTs/Ads/AutostoreStatus.TcDUT
{attribute 'qualified_only'}
{attribute 'strict'}
TYPE AutostoreStatus :
(
	UNKNOWN := 0,
	ROTATING	:=1,
	READY	:=2
);
END_TYPE

// ---- 02DUTs/Ads/BarcodeVerificationResult.TcDUT
{attribute 'qualified_only'}
{attribute 'strict'}
TYPE BarcodeVerificationResult :
(
	UNVERIFIED 	:= 0,
	VALID		:= 1,
	INVALID		:= 2
);
END_TYPE

// ---- 02DUTs/Ads/ButtonStatus.TcDUT
{attribute 'qualified_only'}
{attribute 'strict'}
TYPE ButtonStatus:
(
        PRESSED := 0,
        RELEASED := 1
);
END_TYPE

// ---- 02DUTs/Ads/EStopStatus.TcDUT
{attribute 'qualified_only'}
{attribute 'strict'}
TYPE EStopStatus:
(
        ENGAGED := 0,
        DISENGAGED := 1
);
END_TYPE

// ---- 02DUTs/Ads/E_SAFETYDOOR.TcDUT
{attribute 'qualified_only'}
{attribute 'strict'}
TYPE E_SAFETYDOOR :
(
	IDLE := 0,
	SAFETY,
	UNLOCKING,
	UNLOCKED,
	LOCKED,
	WAIT_LOCKED,
	WAIT_UNLOCKED,
	REQUEST_LOCK
);
END_TYPE

// ---- 02DUTs/Ads/E_SafetyStates.TcDUT
{attribute 'qualified_only'}
{attribute 'strict'}
TYPE E_SafetyStates :
(
	IDLE := 0,
	CHECK_ESTOP,
	CHECK_DOOR_CLOSED,
	CHECK_DOOR_OSSD,
	CHECK_SAFETY_OUTPUT,
	REMIND_RESET,
	DOOR_LOCK,
	TRIG_RESET,
	DONE,
	ERROR
);
END_TYPE

// ---- 02DUTs/Ads/MachineControlCommand.TcDUT
{attribute 'qualified_only'}
{attribute 'strict'}
TYPE MachineControlCommand :
(
	DO_NOTHING  := 0,
	RESET 		:=1,
	START 		:=2,
	STOP 		:=3
);
END_TYPE

// ---- 02DUTs/Ads/MachineStatus.TcDUT
{attribute 'qualified_only'}
{attribute 'strict'}
TYPE MachineStatus:
(
  	STOPPED			:= 0,
   	RESETTING		:= 1,
   	READY			:= 2,
   	INITIALIZING	:= 3,
 	RUNNING			:= 4,
    STOPPING		:= 5,
   	ERROR			:= 6
);
END_TYPE

// ---- 02DUTs/Ads/OrderToteCommand.TcDUT
{attribute 'qualified_only'}
{attribute 'strict'}
TYPE OrderToteCommand:
(
DO_NOTHING	:=0,
LOAD		:=1,
UNLOAD		:=2,
SWAP		:=3,
OPEN_BAG	:=4,
STOP		:=5
);
END_TYPE

// ---- 02DUTs/Ads/OrderToteErrorStatus.TcDUT
{attribute 'qualified_only'}
{attribute 'strict'}
TYPE OrderToteErrorStatus:
(
	UNKNOWN							:=0,
  	NO_ERROR						:=1,
	MACHINE_NOT_RUNNING				:=2,
	ELECTRICAL_ERROR				:=3,
 	MECHANICAL_ERROR				:=4,
 	SAFETY_ERROR					:=5,
	UPSTREAM_NOT_READY				:=6,
	TIMEOUT_WAITING_FOR_NEW_TOTE	:=7,
	DOWNSTREAM_NOT_READY			:=8,
	TIMEOUT_WAITING_FOR_SPACE		:=9
);
END_TYPE

// ---- 02DUTs/Ads/SafetyDoorStatus.TcDUT
{attribute 'qualified_only'}
{attribute 'strict'}
TYPE SafetyDoorStatus:
(
        UNLOCKED := 0,
        LOCKED := 1
);
END_TYPE

// ---- 02DUTs/Ads/SafetyStatus.TcDUT
{attribute 'qualified_only'}
{attribute 'strict'}
TYPE SafetyStatus :
(
	UNKNOWN := 0,
	READY	:=1,
	SAFETY_STOPPED	:=2,
	ERROR	:=3
	
);
END_TYPE

// ---- 02DUTs/Ads/StationMode.TcDUT
{attribute 'qualified_only'}
{attribute 'strict'}
TYPE StationMode :
(
	UNKNOW 			:= 0,
	RUNNING			:= 1,
	RESETTING		:= 2,
	STOPPED			:= 3,
	DISABLED		:= 4,
	STARTING		:= 5,
	FORCE_STOP		:= 6,
	INTERVENTION	:= 7
	
	
);
END_TYPE

// ---- 02DUTs/Ads/ST_LightTower.TcDUT
TYPE ST_LightTower :
STRUCT
	GREEN	: BOOL;
	RED		: BOOL;
	YELLOW	: BOOL;
	BLUE	: BOOL;
	WHITE	: BOOL;
	BUZZER	: BOOL;
END_STRUCT
END_TYPE

// ---- 02DUTs/Ads/ToteStatus.TcDUT
{attribute 'qualified_only'}
{attribute 'strict'}
TYPE ToteStatus:
(
	UNKNOWN 	:= 0,
	EMPTY 		:= 1,
	LOADED		:= 2,
    READY		:= 3
);
END_TYPE

// ---- 02DUTs/Ads/ToteSubsystemWorkflowStatus.TcDUT
{attribute 'qualified_only'}
{attribute 'strict'}
TYPE ToteSubsystemWorkflowStatus:
(
	UNKNOWN					:=0,
  	IDLE					:=1,
 	WAITING_FOR_NEW_TOTE	:=2,
 	INBOUNDING				:=3,
  	BAG_OPENING				:=4,
   	WAITING_FOR_UNLOADING	:=5,
  	OUTBOUNDING				:=6
);
END_TYPE

// ---- Mian/machine/axis/ST_MotionAxis_MC.TcDUT
TYPE ST_MotionAxis_MC :
STRUCT
	rVelocity						: 	LREAL   						;
	rVelocity2						: 	LREAL   						;
	rMaxVelocity					:	LREAL							;	
	rAcceleration					:	LREAL							;
	rMaxAcceleration				:	LREAL							;
	rDeceleration					:	LREAL   						;
	rMaxDeceleration				:	LREAL							;
	rJerk							:	LREAL							;
	rMaxJerk						:	LREAL							;
	rPosition						:	LREAL							;
	rSetPosDistance					:	LREAL							;
	rSetPos							: 	LREAL							;	
	rDistance						:   LREAL							;
	rDistance2						:   LREAL							;	
	
	rActualPosSet					:	LREAL							;//ADD BY EVAN 
	rVelocitySet					: 	LREAL   						;//ADD BY EVAN 	
	xHoming							:	BOOL							;//ADD BY EVAN 
	
	rMaxDistance					:	LREAL							;
	bLimit							:   BOOL							;
	bNegLim							:   BOOL							;
	bPosLim							:	BOOL							;
	bNegSen							:   BOOL							;
	bPosSen							:	BOOL							;
	bPositionSensor					:	BOOL							;
	rHomePos						:	LREAL							;
	rActualPos						:	LREAL							;
	PosDiff							:	LREAL							;
	rActualCurr						:	LREAL							;
	axisDirection					:	MC_Direction					;
	
	rVeloPers						: 	LREAL							;
	rAccPers						: 	LREAL							;   
	rDecPers						: 	LREAL							;                                             					
	SetHomePos						: 	LREAL							;
	HomeVelo						: 	LREAL							;
	PosDiffTarget					: 	LREAL							;
	rFirstpos						: 	LREAL							;
	iAxisID							:	INT								;
	xhsHomingStart					: 	BOOL							;
	xHomingDone						: 	BOOL							;
	xForceControlStart				: 	BOOL							;
	xFoceControlDone				:	BOOL							;	
	xMoveABSDone					: 	BOOL							;
	xMoveRelDone					:	BOOL							;
	bInCouple						:	BOOL							;//Flag Axis is coupled 
    xMuteAxisErrorMessages			:	BOOL							;                                         					
	//Visible/Hide HMI interfaces                   					
	bHomeButtonShow					:	BOOL							; 
	bNegSensorShow					:	BOOL							; 
	bPosSensorShow					:	BOOL							;
	bBacklashShow					:	BOOL							;
	bUnitDegShow					:	BOOL							;
    bJerkShow						:	BOOL							; 
	bStopButtonShow					:	BOOL							; 
	   
	
	bMoveAbsHMI						:	BOOL;
	rVelocityHMI 					: 	LREAL;
	rActualPosHMI					:	LREAL							;//ADD BY EVAN
	bMChomingEnable					:	BOOL							;                                         				
	// backlash compensation                        	
	rBacklashvalue					:	LREAL							;
	xbacklashEnable					:	BOOL							;                        		                					
	bdirFW							:	BOOL							;// on hard stop homing , define the direction of rotation
	
	ModOp					 		: 	SINT							;// Axis operation mode (8 )

//	==============================	Beckhoff Tc2_MC2 library(motion)	==================================
	mcPower 						: 	MC_Power					    ;(*	Axis power, enable/disable																			*)
	mcAxisStates					:	MC_AxisStates					;(*	Driver Feedback, curr motor stage 																	*)
	mcHalt							: 	MC_Halt							;(*	Stops an axis with a defined braking ramp															*)
	mcHome							: 	MC_Home							;(*	Axis homing scenario and execution																	*)
	mcJog							: 	MC_Jog							;(*	Axis Joging BW/FW																					*)	
	mcMoveAbsolute					: 	MC_MoveAbsolute					;(*	Axis GoTo Absolute position																			*)	
	mcMoveRelative					: 	MC_MoveRelative					;(*	Axis GoTo Step by SetPos +/- actual position														*)
	mcMoveVelocity					: 	MC_MoveVelocity					;(*	Axis GoTo with constant velocity														*)
	mcReadStatus					: 	MC_ReadStatus					;(*	Read Axis statuses from driver																		*)
	mcReset							: 	MC_Reset						;(*	Reset Driver																						*)
	mcStop							: 	MC_Stop							;(*	Stop Driver																							*)
	mcReadActualPosition			:	MC_ReadActualPosition			;(*	Read the current axis position																		*)
	mcSetpoint						: 	MC_SetPosition					;(*	Sets the current axis position to a parameterizable value											*)
	mcWriteBoolParameter			: 	MC_WriteBoolParameter			;(*	Write bool param to driver																			*)
	mcReadBoolParameter				:	MC_ReadBoolParameter			;(*	Read bool param from driver																			*)
	mcAxisParameter					:   MC_AxisParameter				;(*	Data type is used in conjunction with function blocks for reading and writing of axis parameters	*)
	CoeWrt							:	FB_EcCoESdoWrite;									
	
//	======================================================================================================	

//
	iSdoWrite	:INT; //6:clear encoder
	sNetID : STRING;
	nSlaveAddr	:UINT;
	nSubIndex	: BYTE;
	nIndex	: WORD;
	
	iCoeWrt	: INT;
	rToqueLimitSet	: LREAL	:= 350;
	rActTorque	: LREAL;
	xTorqueErr	: BOOL;
	iAxis	: WORD;
END_STRUCT
END_TYPE

// ---- Mian/machine/bufferr module/E_RollerStates.TcDUT
{attribute 'qualified_only'}
{attribute 'strict'}
TYPE E_RollerStates :
(
	IDLE := 0,
	INIT,
	DETECTION,
	LOADING,
	UNLOADING,
	STOPPER_DOWN,
	STOPPER_UP,
	ROLLER_FORWARD,
	WAIT_MUTE_OFF,
	UNLOAD_LIFT_MODULE,
	AGING_STATE_0,
	AGING_STATE_1,
	WAIT,
	WAIT_1,
	DONE,
	ERROR
);
END_TYPE

// ---- Mian/machine/bufferr module/Inbound_roller.TcDUT
TYPE Inbound_roller :
STRUCT
	roller : ARRAY[0..1] OF Roller;
	photo_sensor	: ARRAY[0..1] OF BOOL;//[1] light curtain mute
	mcAxis			: FB_MotionAxis_MC;
	st_mcAxis 		: ST_MotionAxis_MC;
	AxisRef			: AXIS_REF;
END_STRUCT
END_TYPE

// ---- Mian/machine/loading moudle/E_LoadingStates.TcDUT
{attribute 'qualified_only'}
{attribute 'strict'}
TYPE E_LoadingStates :
(
	IDLE := 0,
	INIT,
	CHECK,
	WAIT,
	WAIT_1,
	DETECTION,
	LOADING,
	UNLOADING,
	WAIT_NEXT_READY,
	LIFT_POSITION_LOAD,
	LIFT_POSITION_UNLOAD,
	LIFT_UP,
	ROLLER_LOAD,
	ROLLER_UNLOAD,
	WAIT_LEFT_MUTE_OFF,
	WAIT_RIGHT_MUTE_OFF,
	AGING_STATE_0,
	AGING_STATE_1,
	DONE,
	ERROR
);
END_TYPE

// ---- Mian/machine/loading moudle/E_Transfer.TcDUT
{attribute 'qualified_only'}
{attribute 'strict'}
TYPE E_Transfer :
(
	IDLE := 0,
	LOAD,
	UNLOAD
);
END_TYPE

// ---- Mian/machine/loading moudle/Roller_x.TcDUT
TYPE Roller_x :
STRUCT
	
	roller	: Roller;
	photo_sensor_mute_left	 : FB_DigitalInput;
	photo_sensor_mute_right	: FB_DigitalInput;
END_STRUCT
END_TYPE

// ---- Mian/machine/loading moudle/Roller_y.TcDUT
TYPE Roller_y :
STRUCT
	roller	: Roller;
	photo_sensor	: ARRAY[0..1] OF BOOL;
END_STRUCT
END_TYPE

// ---- Mian/machine/mcp/ST_safetyDoor.TcDUT
TYPE ST_safetyDoor :
STRUCT
	button_reset		: BOOL;
	button_unlock		: BOOL;
	door_closed	: BOOL;
	
	lamp_reset			: BOOL;
	lamp_unlock			: BOOL;
	door_lock			: BOOL;
END_STRUCT
END_TYPE

// ---- Mian/machine/Roller.TcDUT
TYPE Roller :
STRUCT
	Power  			: BOOL;
	forward  		: BOOL; 
	backward		: BOOL;
	err 			: BOOL;
	sensor 			: FB_DigitalInput;
END_STRUCT
END_TYPE

// ---- Mian/machine/working moudle/Estates/E_Condition.TcDUT
{attribute 'qualified_only'}
{attribute 'strict'}
TYPE E_Condition :
(
	IDLE 				:= 0,
	PLACE_MOUDULE_UP	:= 1,
	PLACE_MOUDULE_DOWN	:= 2,
	BAG_OPENED			:= 3,
	BAG_CLOSED			:= 4,
	NO_TOTE				:= 5,
	TOTE_IN				:= 6,
	READY_LOADING_TOTE	:= 7
	
);
END_TYPE

// ---- Mian/machine/working moudle/Estates/E_WorkingStates.TcDUT
{attribute 'qualified_only'}
{attribute 'strict'}
TYPE E_WorkingStates ://can't divide into 2 states for load and unload,for sometimes if not unload,then call load,can cause accident
(
	IDLE := 0,
	INIT,
	CHECK,
	WAIT_NEW_TOTE,
	LOADING,
	WAIT_FINISHED,
	TOTE_LOAD,
	TOTE_UNLOAD,
	BAG_OPEN,
	BAG_CLOSE,
	TOTE_LIFT_UP,
	TOTE_LIFT_DOWN,
	BAG_OPEN_UP,
	BAG_OPEN_DOWN,
	TOTE_OUT,
	WAIT_1,
	
	
	BAG_OPEN_HOME,//CYLINDER AND AXIS HOME
	BAG_OPEN_VACUUN_BEGIN,
	VACUUN_ON,
	VACUUN_OFF,
	BAG_OPEN_VACUUN_END,
	BAG_OPEN_SIDE_CYCLINDER_DOWN,
	BAG_OPEN_SIDE_CYCLINDER_UP,
	BAG_OPEN_SIDE_CYCLINDER_EXTEND,
	BAG_OPEN_SIDE_CYCLINDER_RETRACT,
	BAG_OPEN_AXIS_CYCLINDER_DOWN,
	BAG_OPEN_AXIS_CYCLINDER_UP,
	BAG_OPEN_AXIS_CLOSE,
	BAG_OPEN_AXIS_OPEN,
	
	
	AGING_STATE_0,
	AGING_STATE_1,
	
	
	
	
	WAIT,
	
	WAIT_UNLOADING,
	WAIT_SENSOR_ON,
	WAIT_SENSOR_OFF,	
	DONE				:= 100,
	ERROR				:= 200
	
);
END_TYPE

// ---- Mian/machine/working moudle/Inbound.TcDUT
TYPE Inbound :
STRUCT
	roller	: Roller;
	photo_sensor_mute	 : FB_DigitalInput;
	photo_sensor	: FB_DigitalInput;
END_STRUCT
END_TYPE

// ---- Mian/machine/working moudle/Outbound.TcDUT
TYPE Outbound :
STRUCT
	roller	: Roller;
	photo_sensor	: BOOL;
END_STRUCT
END_TYPE

// ---- Mian/statemachine/E_SystemManager.TcDUT
{attribute 'qualified_only'}
{attribute 'strict'}
TYPE E_SystemManager :
(
	START 					:= 0		,	// Solid YELLOW
	ON_POWER 				:= 10		,	// Solid YELLOW
	
	RESET_SAFETY,
	RESET_FB_LOADING,
	RESET_FB_BUFFER,
	RESET_FB_WORKING,
	
	INIT_SAFETY,
	INIT_FB_LOADING,
	INIT_FB_BUFFER,
	INIT_FB_WORKING,
	AGAING_TEST,
	
	READY					:= 	20		,	// Blinking Green
	READY_TO_JOB			:= 	50		,	// Blinking Green
	INITIALIZATION			:= 	100		,	// Blinking YELLOW
	BUSY					:= 	200		,	// Blinking YELLOW

	RUN_START,
	IN_PROGRESS				:= 	300		, 	// Solid Green
	
	IN_PROGRESS_WAITING		:= 	360		,	// blinking Green/Yellow
					
	
	REJECT					:= 	700		,
	RECOVERY				:= 	880 	,
	ERROR					:= 	900		,	// Solid Red
	ERROR_SAFETY			:=	950		,	// Blinking Red
	ERROR_SAFETY_EX			:=	955		,	// Blinking Red

	RESET					:=	990		,	// Blinking Red/Yellow
	RESET_EX				:=	995			// Blinking Red/Yellow


);
END_TYPE

// ---- GVLs/GVL.TcGVL
{attribute 'qualified_only'}
VAR_GLOBAL
	
	devState AT%I*	: UINT;
	arrPD_IN	 AT%I*	: ARRAY[0..31] OF BYTE;
	arrPD_OUT	 AT%Q*	: ARRAY[0..31] OF BYTE;
	fb_working	: FB_working;
	fb_loading	: FB_loading;
	fb_buffer	: FB_buffer;
	fb_mcp		: FB_mcp;
	working_tote_status	: ToteStatus;
	buffer_tote_status	: ToteStatus;
	loading_tote_status	: ToteStatus;
	
	
	
	status	: MachineStatus := MachineStatus.STOPPED;
	workflow_status	: ToteSubsystemWorkflowStatus := ToteSubsystemWorkflowStatus.UNKNOWN;
	error_status	: OrderToteErrorStatus := OrderToteErrorStatus.UNKNOWN;	
	tote_status	: ToteStatus;
	
	events_alarm	: ARRAY[0..iAlarm_max]OF ST_EVENT;
	event_for_clear	: ST_EVENT;
	


	bAck_pause	: BOOL;//avalible while statemachie is IN_PROGRESS
	bAck_stop	: BOOL;
	//bAck_run	: BOOL;
	//bAck_reset	: BOOL;
	
	bRunning	: BOOL;
	bstopped	: BOOL;

END_VAR
VAR_GLOBAL CONSTANT
	iAlarm_max	:INT	:=19;
END_VAR

// ---- GVLs/GVL_IOLink.TcGVL
//{attribute 'qualified_only'}
VAR_GLOBAL
	 
SI0_0              AT%I*  :BOOL           ;   //eStop1/2_NC1	急停1/2_NC1          
SI0_1              AT%I*  :BOOL           ;   //eStop1/2_NC2	急停1/2_NC2          
SI0_2              AT%I*  :BOOL           ;   //safetyDoor_NC1	门锁_NC1           
SI0_3              AT%I*  :BOOL           ;   //safetyDoor_NC2	门锁_NC2           
SI1_0              AT%I*  :BOOL           ;   //eStop3_NC1	急停3_NC1              
SI1_1              AT%I*  :BOOL           ;   //eStop3_NC2	急停3_NC2              
SI1_2              AT%I*  :BOOL           ;   //	                               
SI1_3              AT%I*  :BOOL           ;   //	                               
SI2_0              AT%I*  :BOOL           ;   //light_curtain_left[0]	安全光栅1-ON1 
SI2_1              AT%I*  :BOOL           ;   //light_curtain_left[1]	安全光栅1-ON2 
SI2_2              AT%I*  :BOOL           ;   //eStop4_NC1	急停按钮4-NC1            
SI2_3              AT%I*  :BOOL           ;   //eStop4_NC2	急停按钮4-NC2            
SI3_0              AT%I*  :BOOL           ;   //light_curtain_right[0]	安全光栅2-ON1
SI3_1              AT%I*  :BOOL           ;   //light_curtain_right[1]	安全光栅2-ON2
SI3_2              AT%I*  :BOOL           ;   //station_detection_NC1	升降推到位检测ON1
SI3_3              AT%I*  :BOOL           ;   //station_detection_NC2	升降推到位检测ON2
SI4_0              AT%I*  :BOOL           ;   //屏蔽光栅_left
SI4_1              AT%I*  :BOOL           ;   //屏蔽光栅_right	                                         
SI4_2              AT%I*  :BOOL           ;   
SI4_3              AT%I*  :BOOL           ;   
	                                         
SO0_0              AT%I*  :BOOL           ;   //EES	机器人EES急停         
SO0_1              AT%I*  :BOOL           ;   //EAS	机器人EAS安全门        
SO0_2              AT%I*  :BOOL           ;   //	                    
SO0_3              AT%I*  :BOOL           ;   //	                    
SO1_0              AT%I*  :BOOL           ;   //24v_sto	滚筒电机急停（24V急停）
SO1_1              AT%I*  :BOOL           ;   //A/B_sto	阻挡步进电机（A/B急停）
SO1_2              AT%I*  :BOOL           ;   //	                    
SO1_3              AT%I*  :BOOL           ;   //	                    
SO2_0              AT%I*  :BOOL           ;   //STO1	伺服STO1          
SO2_1              AT%I*  :BOOL           ;   //STO2	伺服STO2          
SO2_2              AT%I*  :BOOL           ;   //24v_sto	滚筒电机急停（24V急停）
SO2_3              AT%I*  :BOOL           ;   //	                    
SO3_0              AT%I*  :BOOL           ;   //STO1	伺服STO1          
SO3_1              AT%I*  :BOOL           ;   //STO2	伺服STO2          
SO3_2              AT%I*  :BOOL           ;   //24v_sto	滚筒电机急停（24V急停）
SO3_3              AT%I*  :BOOL           ;   //	                                                           
	                                        	 

b_FBerror	AT %I*		:	BOOL;//安全功能块错误
b_CoMerror	AT %I*		:	BOOL;//安全端口错误
	 
b_GroupRun	AT %Q*  	:  BOOL:=1;//安全模块运行
b_ErrorAck	AT %Q*  	:  BOOL;//安全模块错误确认
b_EStopRestart AT %Q* 	:  BOOL;	//安全模块复位 	 
	
bMultingEnable AT %Q* 	:  BOOL;
bShield_light_curtain_Left  	AT %Q*  	:  BOOL ;//屏蔽光栅1
bShield_light_curtain_Right  	AT %Q*  	:  BOOL ;//屏蔽光栅2

SPtop_EDM  	AT %Q*  	:  BOOL ;//急停反馈

robot_eas_edm  	AT %Q*  	:  BOOL ;//机械人门安全反馈

light_STO_EDM              AT %Q*  	:  BOOL ; //升降STO反馈
PickModule_STO_EDM         AT %Q*  	:  BOOL ; //分拣STO反馈
Rolller_belt_STO_EDM       AT %Q*  	:  BOOL ; //滚筒STO反馈

               
 END_VAR

// ---- GVLs/G_HMI.TcGVL
{attribute 'qualified_only'}
VAR_GLOBAL
	iMainFrame 		: INT;
	bReset			: BOOL;
	bRun			: BOOL;
	bStop			: BOOL;
	bPause			: BOOL;
	bInit			: BOOL;
	bAging_test		: BOOL;
END_VAR

// ---- GVLs/G_IO.TcGVL
{attribute 'global_init_slot' := '40600'}
VAR_GLOBAL CONSTANT
	{attribute 'global_init_slot'}
	DiMouduleMAX 			:	INT	:=	10;
	{attribute 'global_init_slot'}
	DOMODULEMAX 			:	INT	:=	10;
END_VAR

VAR_GLOBAL

	
	

	arDI	AT%I*		: ARRAY[0..DiMouduleMAX ] OF ST_IO_16;		//  links to Digital input  Modules 
	arDO	AT%Q*		: ARRAY[0..DOMODULEMAX ] OF ST_IO_16;		//  links to Digital output Modules
   
	
END_VAR

// ---- Mian/MAIN.TcPOU
PROGRAM MAIN
VAR
	
	firstCycle	: BOOL := TRUE;
	fb_Time : FB_LocalSystemTime;
	Temp_str : STRING;
   	
	
	str_state	: STRING;
	application	: FB_Application;
	rtReset		: R_TRIG;
	rtInit		: R_TRIG;
	rtRun		: R_TRIG;
	rtSafety	: R_TRIG;
	
	ton_timeout			: TON;	
	eState				: E_SystemManager	:= E_SystemManager.START;
	eStateTemp			: E_SystemManager	:= E_SystemManager.START;
	iStateTemp			: INT;
	sStateTemp			: STRING;	
	
	

	rtStop_auto_store	: R_TRIG;
	pAutostore_control_cmd	: POINTER TO AutostoreControlCommand;
	bButton				: BOOL;
	ton_button			: TON;
	resetting			: BOOL;
	initializing		: BOOL;
	running				: BOOL;
	
	
	pMachine_status	: POINTER TO MachineStatus;
	pMachine_control_cmd	: POINTER TO MachineControlCommand;
	b_test: BOOL;
	event	: ST_EVENT;
	b_test1: BOOL;
	b_test2: BOOL;
	
	bWriteLog	: BOOL;
END_VAR

//////////////////////////////////////////////////////////timeout//////////////////////////////////////////
iStateTemp	:= eStateTemp;
sStateTemp	:= INT_TO_STRING(iStateTemp);
ton_timeout();
IF eState<>E_SystemManager.START AND eState<>E_SystemManager.ERROR THEN
	IF eStateTemp=eState THEN
		ton_timeout.IN	:=TRUE;
	ELSE
		ton_timeout.IN	:=FALSE;
		eStateTemp	:= eState;	
	END_IF
ELSE
	ton_timeout.IN	:=FALSE;
END_IF
IF ton_timeout.Q THEN	
	ton_timeout.IN	:=FALSE;
	CASE eState OF		
		E_SystemManager.START:
			;	
		
	END_CASE
//	IF eStates<>E_WorkingStates.WAIT_NEW_TOTE AND eStates<>E_WorkingStates.WAIT THEN
//		eStates	:= E_WorkingStates.ERROR;
//	END_IF
	
END_IF


IF firstCycle THEN
	firstCycle := FALSE;
END_IF
pMachine_status	:= ADR(MAIN.application.tote_subsystem.status);
pMachine_control_cmd	:= ADR(MAIN.application.tote_subsystem.machine_control_cmd);
fb_Time(bEnable := TRUE);
Temp_str := Prepare_Date_Time(fb_Time.systemTime);
rtSafety(CLK:=application.safety.xError);
rtReset(CLK:=G_HMI.bReset OR GVL.fb_mcp.st_safety_door.button_reset OR pMachine_control_cmd^=MachineControlCommand.RESET);
rtInit(CLK:=G_HMI.bInit);
rtRun(CLK:=G_HMI.bRun);

IF rtSafety.Q THEN
	eState	:= E_SystemManager.ERROR_SAFETY;
END_IF
(******************************************************************************
State Machine
******************************************************************************)
//error while running than estate=error,if electrical error,trig xerror and estate=error
//reset: xError->false and reset devices
//wait 1s,
CASE eState OF
	E_SystemManager.START:
		;
	E_SystemManager.INITIALIZATION:
		;
	E_SystemManager.RESET:
		eState	:= E_SystemManager.RESET_SAFETY;
	E_SystemManager.RESET_SAFETY:
		IF application.safety.M_reset() THEN
			IF application.safety.xError THEN
				eState	:= E_SystemManager.ERROR_SAFETY;
			ELSE
				eState	:= E_SystemManager.RESET_FB_LOADING;
			END_IF
		END_IF
	E_SystemManager.RESET_FB_LOADING:
		IF GVL.fb_loading.M_reset() THEN
			IF GVL.fb_loading.xError THEN
				eState	:= E_SystemManager.ERROR;
			ELSE
				eState	:= E_SystemManager.RESET_FB_BUFFER;
			END_IF
		END_IF
	E_SystemManager.RESET_FB_BUFFER:
		IF GVL.fb_buffer.M_reset() THEN
			IF GVL.fb_buffer.xError THEN
				eState	:= E_SystemManager.ERROR;
			ELSE
				eState	:= E_SystemManager.RESET_FB_WORKING;
			END_IF
		END_IF		
	E_SystemManager.RESET_FB_WORKING:
		IF GVL.fb_working.M_reset() THEN
			IF GVL.fb_working.xError THEN
				eState	:= E_SystemManager.ERROR;
			ELSE
				eState	:= E_SystemManager.READY;
			END_IF
		END_IF		
		
	E_SystemManager.INIT_SAFETY:
		IF application.safety.M_reset() THEN
			IF application.safety.xError THEN
				eState	:= E_SystemManager.ERROR_SAFETY;
			ELSE
				eState	:= E_SystemManager.INIT_FB_LOADING;
			END_IF
		END_IF
	E_SystemManager.INIT_FB_LOADING:
		IF GVL.fb_loading.M_init() THEN
			IF GVL.fb_loading.xError THEN
				eState	:= E_SystemManager.ERROR;
			ELSE
				eState	:= E_SystemManager.INIT_FB_BUFFER;
			END_IF
		END_IF
	E_SystemManager.INIT_FB_BUFFER:
		IF GVL.fb_buffer.M_init() THEN
			IF GVL.fb_buffer.xError THEN
				eState	:= E_SystemManager.ERROR;
			ELSE
				eState	:= E_SystemManager.INIT_FB_WORKING;
			END_IF
		END_IF		
	E_SystemManager.INIT_FB_WORKING:
		IF GVL.fb_working.M_init() THEN
			IF GVL.fb_working.xError THEN
				eState	:= E_SystemManager.ERROR;
			ELSE
				eState	:= E_SystemManager.RESET_SAFETY;
			END_IF
		END_IF				
		
	E_SystemManager.READY:
		eState	:= E_SystemManager.READY_TO_JOB;//todo add condition to jump to ready_to_job
	E_SystemManager.READY_TO_JOB://todo add condition to jump to ready
		pMachine_status^	:= MachineStatus.READY;
		IF G_HMI.bRun OR pMachine_control_cmd^=MachineControlCommand.START THEN
			pMachine_control_cmd^	:= MachineControlCommand.DO_NOTHING;
			GVL.bRunning	:= TRUE;
			eState	:= E_SystemManager.RUN_START;
		END_IF
		IF G_HMI.bAging_test THEN
			eState	:= E_SystemManager.AGAING_TEST;
		END_IF
	E_SystemManager.BUSY:
		;
	E_SystemManager.RUN_START:
		GVL.fb_buffer.M_runStart();
		GVL.fb_loading.M_runStart();
		GVL.fb_working.M_runStart();
		eState	:= E_SystemManager.IN_PROGRESS;
		GVL.bRunning	:= TRUE;
	E_SystemManager.IN_PROGRESS:
		pMachine_status^ := MachineStatus.RUNNING;
		GVL.fb_buffer.M_run();
		GVL.fb_loading.M_run();
		IF pMachine_control_cmd^=MachineControlCommand.STOP OR G_HMI.bStop THEN
			GVL.bRunning	:= FALSE;
			GVL.bAck_stop	:= TRUE;
			pMachine_control_cmd^	:= MachineControlCommand.DO_NOTHING;
		END_IF
		IF GVL.bAck_stop THEN
			IF pMachine_control_cmd^=MachineControlCommand.START OR G_HMI.bRun THEN
				GVL.bRunning	:= TRUE;
				GVL.bAck_stop	:= FALSE;
				pMachine_control_cmd^	:= MachineControlCommand.DO_NOTHING;
			END_IF
		END_IF		
		IF M_checkError() THEN
			GVL.fb_buffer.M_safetyEvent();
			GVL.fb_loading.M_safetyEvent();
			GVL.fb_working.M_safetyEvent();
			eState	:= E_SystemManager.ERROR;
		END_IF
	E_SystemManager.ERROR:
		pMachine_status^	:= MachineStatus.ERROR;
		IF rtReset.Q THEN
			Event_clear();
			pMachine_status^	:= MachineStatus.RESETTING;
			pMachine_control_cmd^	:= MachineControlCommand.DO_NOTHING;
			eState	:= E_SystemManager.RESET_SAFETY;
		END_IF
		IF rtInit.Q THEN
			pMachine_status^	:= MachineStatus.INITIALIZING;
			Event_clear();
			eState	:= E_SystemManager.INIT_SAFETY;					
		END_IF		
	E_SystemManager.ERROR_SAFETY:
		GVL.fb_buffer.M_safetyEvent();
		GVL.fb_loading.M_safetyEvent();
		GVL.fb_working.M_safetyEvent();
		eState	:= E_SystemManager.ERROR;
	E_SystemManager.REJECT:
		; 
	E_SystemManager.ON_POWER://	============================================================================== 
		;							//Check if components and tools ready to state REJECT,else to State ERROR								//check if reject is done then go to ready, else go to error state	
	E_SystemManager.AGAING_TEST:
		GVL.fb_buffer.M_agingTest();
		GVL.fb_loading.M_agingTest();
		//GVL.fb_working.M_agingTest();
END_CASE

IF eState<>E_SystemManager.IN_PROGRESS THEN
	GVL.bAck_stop	:= FALSE;
	GVL.bRunning	:= FALSE;
END_IF
//////////////////////////////////////////////////////////mapping//////////////////////////////////////////
GVL.fb_working(	pre_tote_status:= GVL.fb_loading.current_tote_status);
GVL.fb_loading(	pre_tote_status:=GVL.fb_buffer.fb_rollers[3].current_tote_status,
				next_tote_status:=GVL.fb_working.current_tote_status);
GVL.fb_buffer();
GVL.fb_mcp();
M_convert_estate_string(eState:=eState,str_state=>str_state);

application();



auto_store_simulation();

IF b_test THEN
	event.sTime	:= MAIN.Temp_str;
	event.sComponent_name	:='test';
	event.sEvent_MSG	:='alarm test';
	Event_add(event);
	b_test	:= FALSE;
END_IF
IF b_test1 THEN
	Event_clear();
END_IF
IF bWriteLog THEN
	ADSLOGSTR(msgCtrlMask:= ADSLOG_MSGTYPE_LOG,msgFmtStr:='msg:log',strArg:='MSG ARG');
	bWriteLog	:= FALSE;
END_IF

ACTION auto_store_simulation:

bButton	:= G_IO.arDI[0].Ch[14];
ton_button(IN:=bButton,PT:=T#2S);
pAutostore_control_cmd := ADR(application.tote_subsystem.autostore_control_cmd);
IF ton_button.Q THEN
	pAutostore_control_cmd^	:= AutostoreControlCommand.START;
END_IF
END_ACTION

METHOD M_checkError : BOOL
VAR_INPUT
END_VAR



M_checkError	:= GVL.fb_buffer.xError OR GVL.fb_loading.xError OR GVL.fb_working.xError;
END_METHOD

METHOD M_convert_estate_string : BOOL
VAR_INPUT
	eState	:E_SystemManager;
END_VAR
VAR_OUTPUT
	str_state	: STRING;
END_VAR
CASE eState OF
	E_SystemManager.START:
		str_state	:= 'START';
	E_SystemManager.INITIALIZATION:
		str_state	:= 'INITIALIZATION';
	E_SystemManager.RESET:
		str_state	:= 'RESET';
	E_SystemManager.RESET_SAFETY:
		str_state	:= 'RESET_SAFETY';
	E_SystemManager.RESET_FB_LOADING:
		str_state	:= 'RESET_FB_LOADING';
	E_SystemManager.RESET_FB_BUFFER:
		str_state	:= 'RESET_FB_BUFFER';	
	E_SystemManager.RESET_FB_WORKING:
		str_state	:= 'RESET_FB_WORKING';
	E_SystemManager.INIT_SAFETY:
		str_state	:= 'INIT_SAFETY';
	E_SystemManager.INIT_FB_LOADING:
		str_state	:= 'INIT_FB_LOADING';
	E_SystemManager.INIT_FB_BUFFER:
		str_state	:= 'INIT_FB_BUFFER';
	E_SystemManager.INIT_FB_WORKING:			
		str_state	:= 'INIT_FB_WORKING';		
	E_SystemManager.READY:
		str_state	:= 'READY';
	E_SystemManager.READY_TO_JOB:
		str_state	:= 'READY_TO_JOB';
	E_SystemManager.BUSY:
		str_state	:= 'BUSY';
	E_SystemManager.RUN_START:
		str_state	:= 'RUN_START';
	E_SystemManager.IN_PROGRESS:
		str_state	:= 'IN_PROGRESS';
	E_SystemManager.ERROR:
		str_state	:= 'ERROR';
	E_SystemManager.ERROR_SAFETY:
		str_state	:= 'ERROR_SAFETY';
	E_SystemManager.REJECT:
		str_state	:= 'REJECT';
	E_SystemManager.ON_POWER://	============================================================================== 
		str_state	:= 'ON_POWER';
	E_SystemManager.AGAING_TEST:
		str_state	:= 'AGAING_TEST';
END_CASE
END_METHOD

END_PROGRAM

// ---- 02DUTs/Ads/FB_Application.TcPOU
FUNCTION_BLOCK FB_Application
VAR_INPUT
END_VAR
VAR_OUTPUT
END_VAR
VAR
	safety : FB_Safety_module;
	tote_subsystem	: FB_Tote_Subsystem;
	light_tower	: FB_Light_tower_module;
END_VAR

safety();
light_tower();
tote_subsystem();

GVL.fb_mcp.lightTower := light_tower._lightTower;
GVL.fb_loading.lightTower	:= light_tower._lightTower;

END_FUNCTION_BLOCK

// ---- 02DUTs/Ads/FB_Safety_module.TcPOU
FUNCTION_BLOCK FB_Safety_module
VAR_INPUT
END_VAR
VAR_OUTPUT
END_VAR
VAR
	SI_0	: UINT;
	SI_1	: UINT;
	GI_0 	: UINT;
	GI_1 	: UINT;
	safety_status	: SafetyStatus	:= SafetyStatus.UNKNOWN;
	
	station_mode	: StationMode;
	iStationMode	: UINT;
	iState: INT;
	bEstop_detection	: BOOL;	
	
	ton_timeout	: TON;	
	eStates					:	E_SafetyStates	:=	E_SafetyStates.IDLE;
	iStateTemp			: INT;
	errorMessage	: STRING;
	xError	: BOOL;
	eStates_safetyDoor	: E_SAFETYDOOR	:= E_SAFETYDOOR.IDLE;
	bReset_safetyDoor	: BOOL;
	
	
	
	
	
	GPWM	: FB_GPWM;
	GPWM_1s	: FB_GPWM;
	tonSaftyDelay: TON;
	b_EStopRestarting  : BOOL;
	T_EStopRestart : TON;
//////////////////////SAFETY hardware config///////////////	
	mcp_estop	: BOOL;
	mcp_safetyDoor	: BOOL;
	belt_estop	: BOOL;
	lift_estop : BOOL;
	lift_lightCurtain_left	: BOOL;
	lift_lightCurtain_right	: BOOL;
	lift_station_detection	: BOOL;
	
	robot_EES				: BOOL;
	robot_EAS				: BOOL;
	buffer_safety			: BOOL;
	loading_safety			: BOOL;
	working_safety			: BOOL;
//	buffer_safety_24v		: BOOL;
//	buffer_safety_stepmotor	: BOOL;
//	loding_safety_sto		: BOOL;
//	loding_safety_24v		: BOOL;
//	working_safety_sto		: BOOL;
//	working_safety_24v		: BOOL;
	
	ref_safety_door	: POINTER TO ST_safetyDoor;
	safety_door_unlock_en		: BOOL;
	bStop_button_unlock		: BOOL;//for not receive cmd from tote_subsystem
END_VAR

M_mapping();
M_safetyDoor();
xError	:=NOT(robot_EES AND buffer_safety AND loading_safety AND working_safety); //if only open the door,machine will just stop,so can control the machine munually
//to do:as below commit and reprogram safety project and test

CASE iState	 OF
	0:
	;

	2:
		IF update_station_mode(2) THEN
			iState	:= 0;
		END_IF	
	3:
		IF M_reset() THEN
			iState	:= 0;
		END_IF
		
END_CASE
//安全Safety报警 确认 复位
tonSaftyDelay(IN:= NOT tonSaftyDelay.Q ,PT:=T#1S);
b_ErrorAck := tonSaftyDelay.Q;



GPWM(i_xEnable:=TRUE,i_udiTime:=25,i_udiCycle:=50);
GPWM_1s(i_xEnable:=TRUE,i_udiTime:=500,i_udiCycle:=1000);
//light curtain mute
GVL.fb_working.lightcurtain_mute_left 	:= GVL.fb_buffer.fb_rollers[3].sensor_mute.Q OR GVL.fb_loading.roller_x.photo_sensor_mute_left.Q;   
GVL.fb_working.lightcurtain_mute_right 	:= GVL.fb_loading.roller_x.photo_sensor_mute_right.Q OR GVL.fb_working.roller_inbound.photo_sensor_mute.Q;
 


 //EDM config
 SPtop_EDM  	  	   := TRUE ;  
 robot_eas_edm  	   := TRUE ;
 light_STO_EDM         := TRUE ;
 PickModule_STO_EDM    := TRUE ;
 Rolller_belt_STO_EDM  := TRUE ;

PROPERTY _stationMode : StationMode
GET
_stationMode	:= station_mode;
END_GET
SET
station_mode	:= _stationMode;
END_SET
END_PROPERTY

METHOD M_mapping : BOOL
VAR_INPUT
END_VAR



mcp_estop					:= SI0_0 AND SI0_1;
mcp_safetyDoor				:= SI0_2 AND SI0_3;
belt_estop					:= SI1_0 AND SI1_1;
lift_lightCurtain_left		:= SI2_0 AND SI2_1;
lift_estop					:= SI2_2 AND SI2_3;
lift_lightCurtain_right		:= SI3_0 AND SI3_1;
lift_station_detection		:= SI3_2 AND SI3_3;
bShield_light_curtain_Left	:= SI4_0;
bShield_light_curtain_Right	:= SI4_1;


robot_EES				:= SO0_0;
robot_EAS				:= SO0_1;
buffer_safety			:= SO1_0;

loading_safety			:= SO2_0;

working_safety			:= SO3_0;

	
	                    
                    
                  
	
IF robot_EES AND robot_EAS THEN 
    safety_status := SafetyStatus.READY ;   //正常
ELSE
	safety_status := SafetyStatus.SAFETY_STOPPED; //急停状态
END_IF

GI_0.0	:= GVL.fb_mcp.st_safety_door.button_reset;
GI_0.1	:= GVL.fb_mcp.st_safety_door.button_unlock;
GI_0.2	:= GVL.fb_mcp.st_safety_door.door_closed;

SI_0.0	:= mcp_estop;
SI_0.1	:= mcp_safetyDoor;
SI_0.2	:= belt_estop;
SI_0.3	:= lift_estop;
SI_0.4	:= lift_station_detection;
END_METHOD

METHOD M_reset : BOOL
VAR_INPUT
	
END_VAR
M_reset	:= FALSE;
//check if all estop
//check if safety door ossd
//check if safety door closed
//lock safety door 
//reset to output safety
//////////////////////////////////////////////////////////timeout//////////////////////////////////////////
ton_timeout();
IF eStates<>E_SafetyStates.IDLE AND eStates<>E_SafetyStates.ERROR  THEN
	IF iStateTemp=eStates THEN
		ton_timeout.IN	:=TRUE;
	ELSE
		ton_timeout.IN	:=FALSE;
		iStateTemp	:= eStates;
	END_IF
ELSE
	ton_timeout.IN	:=FALSE;
END_IF
IF ton_timeout.Q THEN	
	ton_timeout.IN	:=FALSE;
	CASE eStates OF
		E_SafetyStates.DOOR_LOCK:		
			errorMessage	:= CONCAT('door lock error.->safety ',INT_TO_STRING(iStateTemp));
	END_CASE
	IF eStates=E_SafetyStates.DOOR_LOCK AND eStates<>E_SafetyStates.TRIG_RESET THEN
		eStates	:= E_SafetyStates.ERROR;
	END_IF
	
END_IF
CASE eStates OF
	E_SafetyStates.IDLE:
		xError	:= FALSE;
		bReset_safetyDoor	:= FALSE;
		eStates	:= E_SafetyStates.CHECK_ESTOP;
	E_SafetyStates.CHECK_ESTOP:
		IF mcp_estop AND belt_estop AND lift_estop THEN
			eStates	:= E_SafetyStates.CHECK_DOOR_CLOSED;
		ELSE
			eStates	:= E_SafetyStates.ERROR;
		END_IF
	E_SafetyStates.CHECK_DOOR_CLOSED:
		IF GVL.fb_mcp.st_safety_door.door_closed THEN
			eStates	:= E_SafetyStates.DOOR_LOCK;
		ELSE
			eStates	:= E_SafetyStates.ERROR;
		END_IF
	E_SafetyStates.DOOR_LOCK:
		bReset_safetyDoor	:= TRUE;
//		ref_safety_door^.door_lock	:= FALSE;
		IF mcp_safetyDoor THEN
			bReset_safetyDoor	:= FALSE;
			eStates	:= E_SafetyStates.TRIG_RESET;
		END_IF		
	E_SafetyStates.TRIG_RESET:
		ton_timeout.PT	:= T#2S;
		b_EStopRestart	:= GPWM.q_xOut;
		IF ton_timeout.Q THEN
			b_EStopRestart	:= FALSE;
			eStates	:= E_SafetyStates.CHECK_SAFETY_OUTPUT;
		END_IF
	E_SafetyStates.CHECK_SAFETY_OUTPUT:	
		IF robot_EES AND robot_EAS AND buffer_safety AND loading_safety AND working_safety THEN
			eStates	:= E_SafetyStates.DONE;
		ELSE
			eStates	:= E_SafetyStates.ERROR;
		END_IF
	E_SafetyStates.DONE:
		M_reset	:= TRUE;
		eStates	:= E_SafetyStates.IDLE;
	E_SafetyStates.ERROR:	
		M_reset	:= TRUE;
		xError	:= TRUE;
		bReset_safetyDoor	:= FALSE;
		eStates	:= E_SafetyStates.IDLE;

	
END_CASE
END_METHOD

METHOD M_safetyDoor : BOOL
VAR_INPUT
	
END_VAR
ref_safety_door	:= ADR(GVL.fb_mcp.st_safety_door);
safety_door_unlock_en	:= (safety_status=SafetyStatus.SAFETY_STOPPED OR station_mode = StationMode.STOPPED OR station_mode = StationMode.DISABLED
							OR station_mode = StationMode.FORCE_STOP OR station_mode = StationMode.INTERVENTION) AND GVL.fb_working.bStopped;

							
CASE eStates_safetyDoor	 OF
	E_SAFETYDOOR.IDLE:
		IF mcp_safetyDoor THEN
			eStates_safetyDoor	:= E_SAFETYDOOR.LOCKED;
		ELSE
			eStates_safetyDoor	:= E_SAFETYDOOR.UNLOCKED;
		END_IF
	E_SAFETYDOOR.LOCKED:
		ref_safety_door^.lamp_reset	:=	FALSE;
		ref_safety_door^.lamp_unlock	:= FALSE;
		IF ref_safety_door^.button_unlock THEN
			bStop_button_unlock	:= TRUE;
			eStates_safetyDoor	:= E_SAFETYDOOR.UNLOCKING;
		END_IF
	E_SAFETYDOOR.REQUEST_LOCK:
	;
	E_SAFETYDOOR.SAFETY:
	;
	E_SAFETYDOOR.UNLOCKED:
		ref_safety_door^.lamp_unlock	:= TRUE;//door unlocked,unlock lamp solid
		IF ref_safety_door^.door_closed THEN
			ref_safety_door^.lamp_reset	:= GPWM_1s.q_xOut;//door closed,reset lamp blinking
			IF ref_safety_door^.button_reset OR bReset_safetyDoor THEN
				bStop_button_unlock	:= FALSE;
				eStates_safetyDoor	:= E_SAFETYDOOR.WAIT_LOCKED;
			END_IF
		ELSE
			ref_safety_door^.lamp_reset	:= FALSE;
		END_IF
	E_SAFETYDOOR.WAIT_LOCKED:
		ref_safety_door^.door_lock	:= FALSE;
		IF mcp_safetyDoor THEN
			eStates_safetyDoor	:= E_SAFETYDOOR.LOCKED;
	 	END_IF
	E_SAFETYDOOR.UNLOCKING:
		ref_safety_door^.lamp_unlock	:= GPWM_1s.q_xOut;//door opennig,unlock lamp blinking
		IF safety_door_unlock_en THEN
			ref_safety_door^.door_lock	:= TRUE;
			IF NOT mcp_safetyDoor THEN
				eStates_safetyDoor	:= E_SAFETYDOOR.UNLOCKED;
			END_IF
		END_IF
	
END_CASE
END_METHOD

{attribute 'TcRpcEnable'}
METHOD update_station_mode  : BOOL
VAR_INPUT
	iMode	: StationMode;
END_VAR
update_station_mode	:= FALSE;
station_mode	:= iMode;
update_station_mode	:= TRUE;
END_METHOD

END_FUNCTION_BLOCK

// ---- Mian/machine/working moudle/FB_working.TcPOU
FUNCTION_BLOCK FB_working
VAR_INPUT
	lightcurtain_mute_left	: BOOL;
	lightcurtain_mute_right	: BOOL;
	pre_tote_status			: ToteStatus;//roller -1 totestatus=ready
	next_tote_status		: ToteStatus;//roller +1 totestatus=empty
END_VAR
VAR_OUTPUT
	status			: MachineStatus := MachineStatus.STOPPED;
	workflow_status	: ToteSubsystemWorkflowStatus := ToteSubsystemWorkflowStatus.UNKNOWN;
	error_status	: OrderToteErrorStatus := OrderToteErrorStatus.UNKNOWN;	
	tote_status		: ToteStatus;
END_VAR
VAR
	current_tote_status	: ToteStatus;
	ton_timeout			: TON;	
	eStates				: E_WorkingStates	:= E_WorkingStates.IDLE;
	eStateTemp			: E_WorkingStates	:= E_WorkingStates.IDLE;
	iStateTemp			: INT;
	sStateTemp			: STRING;
	errorMessage		: STRING;
	xError				: BOOL;
	iMethod_test		: INT;

	xLoading			: BOOL;
	xUnloading			: BOOL;
///////

	valve_lift			: Valve;
	roller_inbound		: Inbound;
	roller_outbound		: Outbound;
	roller_outbound_end	: Outbound;
	sensor_openbag_detection	: ARRAY[0..7] OF BOOL;
	sensor_cover				: ARRAY[0..1] OF BOOL;
	EDM_KA10			: BOOL;
	mcAxis_lift 		: FB_MotionAxis_MC;
	st_mcAxis_lift 		: ST_MotionAxis_MC;
	AxisRef_lift		: AXIS_REF;
	
	mcAxis_bag 		: FB_MotionAxis_MC;
	st_mcAxis_bag		: ST_MotionAxis_MC;
	AxisRef_bag		: AXIS_REF;	
	
	
	mcAxis_vacuun 		: ARRAY[0..1] OF FB_MotionAxis_MC;
	st_mcAxis_vacuun 		: ARRAY[0..1] OF ST_MotionAxis_MC;
	AxisRef_vacuun		: ARRAY[0..1] OF AXIS_REF;	
	mcAxis_bagOpen 		: ARRAY[0..3] OF FB_MotionAxis_MC;
	st_mcAxis_bagOpen 		: ARRAY[0..3] OF ST_MotionAxis_MC;
	AxisRef_bagOpen		: ARRAY[0..3] OF AXIS_REF;	
	
	valve_open_side		: Valve;//4 cylinders
	valve_open_lift		: Valve;//8 cylinders
	valve_vacuun		: ARRAY[0..3] OF Valve;
	bag_open_detection	: ARRAY[0..3]OF FB_DigitalInput;

	
	
	
	
	

	event				: ST_EVENT;
	rt_error			: R_TRIG;
	eTransfer			: E_Transfer;
	
	
	
	
	
	
	
	bStopped				: BOOL;
END_VAR
VAR CONSTANT
	rPos_lift_up			: REAL	:= 120;
	rPos_lift_down			: REAL	:= 7;
	rPos_vacuun_home		: ARRAY[0..1]OF REAL:=[0,0];
	rPos_vacuun_working		: ARRAY[0..1]OF REAL:=[249,242];
	rPos_bag_begin			: ARRAY[0..3]OF REAL:=[10,10,10,10];
	rPos_bag_end			: ARRAY[0..3]OF REAL:=[95,95,95,95];
	
	
	rPos_bag_opened			: REAL	:= 45;
	rPos_bag_closed			: REAL	:= 0;
	sComponent_name			: STRING := 'fb_working';
END_VAR

M_mapping();

rt_error(CLK:=(roller_inbound.roller.err OR roller_outbound.roller.err OR roller_outbound_end.roller.err OR st_mcAxis_lift.mcReadStatus.Error 
				OR st_mcAxis_bag.mcReadStatus.Error) AND MAIN.eState<>E_SystemManager.RESET_SAFETY);//roller will trig error while power on
IF rt_error.Q THEN
	xError	:= TRUE;
	eStates	:= E_WorkingStates.ERROR;
END_IF

IF NOT(roller_inbound.photo_sensor_mute.Q OR roller_inbound.photo_sensor.Q OR roller_outbound.photo_sensor.Q) THEN
	current_tote_status	:= ToteStatus.EMPTY;
END_IF
IF NOT roller_inbound.photo_sensor_mute.Q AND roller_inbound.photo_sensor.Q AND NOT roller_outbound.photo_sensor.Q THEN
	current_tote_status	:= ToteStatus.READY;
END_IF



IF eStates=E_WorkingStates.IDLE THEN
	bStopped	:= TRUE;
ELSE
	bStopped	:= FALSE;
END_IF
CASE iMethod_test OF
	0:
	;
	1:		
		IF 	M_load() THEN
			iMethod_test	:= 0;
		END_IF
	2:
		IF 	M_bag_open() THEN
			iMethod_test	:= 0;
		END_IF
	3:
		IF 	M_unload() THEN
			iMethod_test	:= 0;
		END_IF
		
END_CASE

METHOD M_agingTest : BOOL
VAR_INPUT
	
END_VAR
M_AgingTest	:= FALSE;
//////////////////////////////////////////////////////////timeout//////////////////////////////////////////
iStateTemp	:= eStateTemp;
ton_timeout();
IF eStates<>E_WorkingStates.IDLE AND eStates<>E_WorkingStates.ERROR THEN
	IF eStateTemp=eStates THEN
		ton_timeout.IN	:=TRUE;
	ELSE
		ton_timeout.IN	:=FALSE;
		eStateTemp	:= eStates;
	END_IF
ELSE
	ton_timeout.IN	:=FALSE;
END_IF
IF ton_timeout.Q THEN	
	ton_timeout.IN	:=FALSE;
	CASE eStates OF
		E_WorkingStates.AGING_STATE_0:		
			errorMessage	:= CONCAT('wait loading timeout.->fb_loading ',INT_TO_STRING(iStateTemp));
		E_WorkingStates.AGING_STATE_1:		
			errorMessage	:= CONCAT('wait unloading timeout.->fb_loading ',INT_TO_STRING(iStateTemp));
	END_CASE
	IF eStates<>E_WorkingStates.WAIT AND eStates<>E_WorkingStates.WAIT_1 THEN
		//eStates	:= E_WorkingStates.ERROR;
		;
	END_IF
END_IF
CASE eStates OF
	E_WorkingStates.IDLE:
		eStates	:= E_WorkingStates.AGING_STATE_0;
	E_WorkingStates.AGING_STATE_0:
		ton_timeout.PT	:= T#2S;
		st_mcAxis_bag.mcMoveAbsolute.Execute	:= TRUE;						
		st_mcAxis_bag.rActualPosSet	:= rPos_bag_closed;
		st_mcAxis_bag.rVelocitySet	:= 100;
		st_mcAxis_lift.mcMoveAbsolute.Execute	:= TRUE;	
		st_mcAxis_lift.rActualPosSet	:= rPos_lift_up;
		st_mcAxis_lift.rVelocitySet	:= 100;	
		roller_inbound.roller.forward			:= TRUE;
		roller_inbound.roller.backward			:= FALSE;
		roller_outbound.roller.forward			:= TRUE;
		roller_outbound_end.roller.forward		:= TRUE;
		roller_outbound_end.roller.backward		:= FALSE;			
		IF st_mcAxis_bag.mcMoveAbsolute.Done AND st_mcAxis_lift.mcMoveAbsolute.Done AND ton_timeout.Q THEN
			eStates	:= E_WorkingStates.WAIT;
		END_IF			
	E_WorkingStates.WAIT:
		roller_inbound.roller.forward			:= FALSE;
		roller_inbound.roller.backward			:= FALSE;
		roller_outbound.roller.forward			:= FALSE;
		roller_outbound.roller.backward			:= FALSE;
		roller_outbound_end.roller.forward		:= FALSE;
		roller_outbound_end.roller.backward		:= FALSE;	
		st_mcAxis_bag.mcMoveAbsolute.Execute	:= FALSE;
		st_mcAxis_lift.mcMoveAbsolute.Execute	:= FALSE;		
		ton_timeout.PT	:= T#1S;
		IF ton_timeout.Q THEN
			eStates	:= E_WorkingStates.AGING_STATE_1;
		END_IF
	E_WorkingStates.AGING_STATE_1:
		ton_timeout.PT	:= T#2S;
		st_mcAxis_bag.mcMoveAbsolute.Execute	:= TRUE;						
		st_mcAxis_bag.rActualPosSet	:= rPos_bag_opened;
		st_mcAxis_bag.rVelocitySet	:= 100;
		st_mcAxis_lift.mcMoveAbsolute.Execute	:= TRUE;
		st_mcAxis_lift.rActualPosSet	:= rPos_lift_down;
		st_mcAxis_lift.rVelocitySet	:= 100;	
		roller_inbound.roller.forward			:= TRUE;
		roller_inbound.roller.backward			:= TRUE;
		roller_outbound.roller.backward			:= TRUE;
		roller_outbound_end.roller.forward		:= TRUE;
		roller_outbound_end.roller.backward		:= TRUE;			
		IF st_mcAxis_bag.mcMoveAbsolute.Done AND st_mcAxis_lift.mcMoveAbsolute.Done AND ton_timeout.Q THEN
			eStates	:= E_WorkingStates.WAIT_1;
		END_IF	
	E_WorkingStates.WAIT_1:
		ton_timeout.PT	:= T#1S;
		roller_inbound.roller.forward			:= FALSE;
		roller_inbound.roller.backward			:= FALSE;
		roller_outbound.roller.forward			:= FALSE;
		roller_outbound.roller.backward			:= FALSE;
		roller_outbound_end.roller.forward		:= FALSE;
		roller_outbound_end.roller.backward		:= FALSE;	
		st_mcAxis_bag.mcMoveAbsolute.Execute	:= FALSE;
		st_mcAxis_lift.mcMoveAbsolute.Execute	:= FALSE;		
		IF ton_timeout.Q THEN
			eStates	:= E_WorkingStates.IDLE;
		END_IF		
	E_WorkingStates.DONE:
		;
	E_WorkingStates.ERROR:
		;
	
END_CASE
END_METHOD

METHOD M_bag_close : BOOL
VAR_INPUT
END_VAR
END_METHOD

METHOD M_bag_open : BOOL
VAR_INPUT
END_VAR
M_bag_open	:= FALSE;
ADSLOGSTR(msgCtrlMask:= ADSLOG_MSGTYPE_LOG,msgFmtStr:='bag open',strArg:='MSG ARG');
M_bag_open	:= TRUE;
END_METHOD

METHOD M_checkCondition : BOOL
VAR_INPUT
	condition	: E_Condition;
END_VAR
M_checkCondition	:= FALSE;
CASE condition OF
	E_Condition.NO_TOTE:
	 	IF NOT roller_inbound.photo_sensor.Q THEN
			M_checkCondition	:= TRUE;
		END_IF
	E_Condition.TOTE_IN:
	 	IF roller_inbound.photo_sensor.Q THEN
			M_checkCondition	:= TRUE;
		END_IF		
	E_Condition.READY_LOADING_TOTE:
		IF pre_tote_status=ToteStatus.READY THEN
			M_checkCondition	:= TRUE;
		END_IF
	E_Condition.TOTE_READY:
		IF ABS(st_mcAxis_lift.mcReadActualPosition.Position-rPos_lift_down)<1 
		AND ABS(st_mcAxis_vacuun[0].mcReadActualPosition.Position-rPos_vacuun_working[0])<1 
		AND ABS(st_mcAxis_vacuun[1].mcReadActualPosition.Position-rPos_vacuun_working[1])<1 
		AND ABS(st_mcAxis_bagOpen[0].mcReadActualPosition.Position-rPos_bag_end[0])<1 
		AND ABS(st_mcAxis_bagOpen[1].mcReadActualPosition.Position-rPos_bag_end[1])<1 
		AND ABS(st_mcAxis_bagOpen[2].mcReadActualPosition.Position-rPos_bag_end[2])<1 
		AND ABS(st_mcAxis_bagOpen[3].mcReadActualPosition.Position-rPos_bag_end[3])<1 
		AND roller_inbound.photo_sensor.Q AND NOT roller_inbound.photo_sensor_mute.Q 
		AND NOT roller_outbound.photo_sensor.Q AND valve_lift.retracted THEN
			tote_status	:= ToteStatus.READY;
		ELSE
			IF tote_status = ToteStatus.READY THEN
				tote_status	:= ToteStatus.LOADED;
			END_IF
		END_IF
		IF ABS(st_mcAxis_lift.mcReadActualPosition.Position-rPos_lift_up)<1 
		AND ABS(st_mcAxis_vacuun[0].mcReadActualPosition.Position-rPos_vacuun_working[0])<1 
		AND ABS(st_mcAxis_vacuun[1].mcReadActualPosition.Position-rPos_vacuun_working[1])<1 
		AND ABS(st_mcAxis_bagOpen[0].mcReadActualPosition.Position-rPos_bag_begin[0])<1 
		AND ABS(st_mcAxis_bagOpen[1].mcReadActualPosition.Position-rPos_bag_begin[1])<1 
		AND ABS(st_mcAxis_bagOpen[2].mcReadActualPosition.Position-rPos_bag_begin[2])<1 
		AND ABS(st_mcAxis_bagOpen[3].mcReadActualPosition.Position-rPos_bag_begin[3])<1 
		AND NOT roller_inbound.photo_sensor.Q AND NOT roller_inbound.photo_sensor_mute.Q
	 	AND NOT roller_outbound.photo_sensor.Q AND valve_lift.retracted THEN
			tote_status	:= ToteStatus.EMPTY;	
		END_IF	
		M_checkCondition	:= TRUE;
END_CASE
END_METHOD

METHOD M_init : BOOL
VAR_INPUT
END_VAR
M_init	:= FALSE;
event.sMethod	:= 'init';
xError	:= FALSE;


st_mcAxis_lift.mcStop.Execute	:= FALSE;
st_mcAxis_vacuun[0].mcStop.Execute	:= FALSE;
st_mcAxis_vacuun[1].mcStop.Execute	:= FALSE;
st_mcAxis_bagOpen[0].mcStop.Execute	:= FALSE;
st_mcAxis_bagOpen[1].mcStop.Execute	:= FALSE;
st_mcAxis_bagOpen[2].mcStop.Execute	:= FALSE;
st_mcAxis_bagOpen[3].mcStop.Execute	:= FALSE;	
st_mcAxis_lift.mcReset.Execute			:= TRUE;
st_mcAxis_vacuun[0].mcReset.Execute		:= TRUE;
st_mcAxis_vacuun[1].mcReset.Execute		:= TRUE;
st_mcAxis_bagOpen[0].mcReset.Execute	:= TRUE;
st_mcAxis_bagOpen[1].mcReset.Execute	:= TRUE;
st_mcAxis_bagOpen[2].mcReset.Execute	:= TRUE;
st_mcAxis_bagOpen[3].mcReset.Execute	:= TRUE;
error_status	:= OrderToteErrorStatus.NO_ERROR;

eStates	:= E_WorkingStates.IDLE;
M_init	:= TRUE;
END_METHOD

METHOD M_load : BOOL
VAR_INPUT
END_VAR
VAR_OUTPUT 

END_VAR
M_load := FALSE;
event.sMethod	:= 'load';
//////////////////////////////////////////////////////////timeout//////////////////////////////////////////
iStateTemp	:= eStateTemp;
sStateTemp	:= INT_TO_STRING(iStateTemp);
ton_timeout();
IF eStates<>E_WorkingStates.IDLE AND eStates<>E_WorkingStates.ERROR THEN
	IF eStateTemp=eStates THEN
		ton_timeout.IN	:=TRUE;
	ELSE
		ton_timeout.IN	:=FALSE;
		IF GVL.bAck_stop THEN
			roller_inbound.roller.forward	:= FALSE;
			RETURN;			
		END_IF
		eStateTemp	:= eStates;	
	END_IF
ELSE
	ton_timeout.IN	:=FALSE;
END_IF
IF ton_timeout.Q THEN	
	ton_timeout.IN	:=FALSE;
	CASE eStates OF		
		E_WorkingStates.BAG_OPEN_UP:	
			event.sEventType	:= 'error';
			event.sEvent_MSG	:= CONCAT('BAG_OPEN_UP ','timeout');
			event.sStepID		:= sStateTemp;
		E_WorkingStates.BAG_CLOSE:	
			event.sEventType	:= 'error';
			event.sEvent_MSG	:= CONCAT('BAG_CLOSE ','timeout');
			event.sStepID		:= sStateTemp;					
		E_WorkingStates.TOTE_LIFT_DOWN:			
			event.sEventType	:= 'error';
			event.sEvent_MSG	:= CONCAT('TOTE_LIFT_DOWN ','timeout');
			event.sStepID		:= sStateTemp;
		E_WorkingStates.WAIT_NEW_TOTE://wait empty and trig signal
			;
		E_WorkingStates.TOTE_LOAD:	
			event.sEventType	:= 'error';
			event.sEvent_MSG	:= CONCAT('TOTE_LOAD ','timeout');
			event.sStepID		:= sStateTemp;
		E_WorkingStates.WAIT:
			;
		E_WorkingStates.BAG_OPEN_DOWN:
			event.sEventType	:= 'error';
			event.sEvent_MSG	:= CONCAT('BAG_OPEN_DOWN ','timeout');
			event.sStepID		:= sStateTemp;			
		E_WorkingStates.BAG_OPEN:			
			event.sEventType	:= 'error';
			event.sEvent_MSG	:= CONCAT('BAG_OPEN ','timeout');
			event.sStepID		:= sStateTemp;
		ELSE
			event.sEventType	:= 'error';
			event.sEvent_MSG	:= CONCAT('unknow estate ','timeout');
			event.sStepID		:= sStateTemp;			
	END_CASE
	IF eStates<>E_WorkingStates.WAIT_NEW_TOTE AND eStates<>E_WorkingStates.WAIT AND eStates<>E_WorkingStates.BAG_OPEN_AXIS_CYCLINDER_DOWN
	AND eStates<>E_WorkingStates.VACUUN_ON AND eStates<>E_WorkingStates.WAIT_1 THEN
		eStates	:= E_WorkingStates.ERROR;
		error_status	:= OrderToteErrorStatus.MECHANICAL_ERROR;
		Event_add(event);
	END_IF
	
END_IF

CASE eStates OF 
		E_WorkingStates.IDLE:
			
			ton_timeout.PT	:= T#10S;
			xLoading	:= FALSE;
			xUnloading	:= FALSE;

			st_mcAxis_vacuun[0].mcPower.Enable	:= TRUE;	
			st_mcAxis_vacuun[1].mcPower.Enable	:= TRUE;
			st_mcAxis_bagOpen[0].mcPower.Enable	:= TRUE;
			st_mcAxis_bagOpen[1].mcPower.Enable	:= TRUE;
			st_mcAxis_bagOpen[2].mcPower.Enable	:= TRUE;
			st_mcAxis_bagOpen[3].mcPower.Enable	:= TRUE;
			st_mcAxis_lift.mcPower.Enable	:= TRUE;
			IF st_mcAxis_vacuun[0].mcReadStatus.StandStill AND st_mcAxis_vacuun[1].mcReadStatus.StandStill AND st_mcAxis_bagOpen[0].mcReadStatus.StandStill
			AND st_mcAxis_bagOpen[1].mcReadStatus.StandStill AND st_mcAxis_bagOpen[2].mcReadStatus.StandStill AND st_mcAxis_bagOpen[3].mcReadStatus.StandStill 
			AND st_mcAxis_lift.mcReadStatus.StandStill THEN
				eStates	:= E_WorkingStates.INIT;
			END_IF			
		E_WorkingStates.INIT:
			ADSLOGSTR(msgCtrlMask:= ADSLOG_MSGTYPE_LOG,msgFmtStr:='load start',strArg:='');
			xLoading	:= TRUE;		
			st_mcAxis_vacuun[0].mcMoveAbsolute.Execute	:= FALSE;
			st_mcAxis_vacuun[1].mcMoveAbsolute.Execute	:= FALSE;
			st_mcAxis_bagOpen[0].mcMoveAbsolute.Execute	:= FALSE;
			st_mcAxis_bagOpen[1].mcMoveAbsolute.Execute	:= FALSE;
			st_mcAxis_bagOpen[2].mcMoveAbsolute.Execute	:= FALSE;
			st_mcAxis_bagOpen[3].mcMoveAbsolute.Execute	:= FALSE;
			valve_open_lift.extend	:= FALSE;
			valve_open_lift.retract	:= TRUE;
			valve_open_side.extend	:= FALSE;
			valve_open_side.retract	:= TRUE;
			valve_vacuun[0].extend	:= FALSE;
			valve_vacuun[0].retract	:= TRUE;
			valve_vacuun[1].extend	:= FALSE;
			valve_vacuun[1].retract	:= TRUE;
			valve_vacuun[2].extend	:= FALSE;
			valve_vacuun[2].retract	:= TRUE;
			valve_vacuun[3].extend	:= FALSE;
			valve_vacuun[3].retract	:= TRUE;			
			st_mcAxis_lift.mcMoveAbsolute.Execute	:= FALSE;
			eStates	:= E_WorkingStates.BAG_OPEN_UP;
		E_WorkingStates.BAG_OPEN_UP:	
			st_mcAxis_lift.mcMoveAbsolute.Execute	:= TRUE;		
			st_mcAxis_lift.rActualPosSet	:= rPos_lift_up;
			st_mcAxis_lift.rVelocitySet	:= 250;
			IF st_mcAxis_lift.mcMoveAbsolute.Done THEN
				st_mcAxis_lift.mcMoveAbsolute.Execute	:= FALSE;
				eStates	:= E_WorkingStates.BAG_OPEN_HOME;
			END_IF	
		E_WorkingStates.BAG_OPEN_HOME:	
			st_mcAxis_vacuun[0].mcMoveAbsolute.Execute	:= TRUE;		
			st_mcAxis_vacuun[0].rActualPosSet	:= rPos_vacuun_working[0];
			st_mcAxis_vacuun[0].rVelocitySet	:= 450;
			st_mcAxis_vacuun[1].mcMoveAbsolute.Execute	:= TRUE;		
			st_mcAxis_vacuun[1].rActualPosSet	:= rPos_vacuun_working[1];
			st_mcAxis_vacuun[1].rVelocitySet	:= 450;			
			st_mcAxis_bagOpen[0].mcMoveAbsolute.Execute	:= TRUE;		
			st_mcAxis_bagOpen[0].rActualPosSet	:= rPos_bag_begin[0];
			st_mcAxis_bagOpen[0].rVelocitySet	:= 200;			
			st_mcAxis_bagOpen[1].mcMoveAbsolute.Execute	:= TRUE;		
			st_mcAxis_bagOpen[1].rActualPosSet	:= rPos_bag_begin[1];
			st_mcAxis_bagOpen[1].rVelocitySet	:= 200;				
			st_mcAxis_bagOpen[2].mcMoveAbsolute.Execute	:= TRUE;		
			st_mcAxis_bagOpen[2].rActualPosSet	:= rPos_bag_begin[2];
			st_mcAxis_bagOpen[2].rVelocitySet	:= 200;				
			st_mcAxis_bagOpen[3].mcMoveAbsolute.Execute	:= TRUE;		
			st_mcAxis_bagOpen[3].rActualPosSet	:= rPos_bag_begin[3];
			st_mcAxis_bagOpen[3].rVelocitySet	:= 200;				
			
			IF st_mcAxis_vacuun[0].mcMoveAbsolute.Done AND st_mcAxis_vacuun[1].mcMoveAbsolute.Done AND st_mcAxis_bagOpen[0].mcMoveAbsolute.Done
			AND st_mcAxis_bagOpen[1].mcMoveAbsolute.Done AND st_mcAxis_bagOpen[2].mcMoveAbsolute.Done AND st_mcAxis_bagOpen[3].mcMoveAbsolute.Done THEN
				st_mcAxis_vacuun[0].mcMoveAbsolute.Execute	:= FALSE;
				st_mcAxis_vacuun[1].mcMoveAbsolute.Execute	:= FALSE;
				st_mcAxis_bagOpen[0].mcMoveAbsolute.Execute	:= FALSE;
				st_mcAxis_bagOpen[1].mcMoveAbsolute.Execute	:= FALSE;
				st_mcAxis_bagOpen[2].mcMoveAbsolute.Execute	:= FALSE;
				st_mcAxis_bagOpen[3].mcMoveAbsolute.Execute	:= FALSE;
				eStates	:= E_WorkingStates.TOTE_LIFT_DOWN;
			END_IF					
		E_WorkingStates.TOTE_LIFT_DOWN:			
			valve_lift.extend	:= FALSE;
			valve_lift.retract	:= TRUE;
			IF NOT valve_lift.extended AND valve_lift.retracted THEN
				eStates	:= E_WorkingStates.WAIT_NEW_TOTE;
			END_IF	
		E_WorkingStates.WAIT_NEW_TOTE://wait empty and trig signal
			workflow_status	:= ToteSubsystemWorkflowStatus.WAITING_FOR_NEW_TOTE;
			IF NOT(roller_inbound.photo_sensor_mute.Q OR roller_inbound.photo_sensor.Q OR roller_outbound.photo_sensor.Q) THEN
				tote_status	:= ToteStatus.EMPTY;
			END_IF
			IF M_waitCondition(condition:=E_Condition.READY_LOADING_TOTE) THEN
				eStates	:= E_WorkingStates.TOTE_LOAD;
			END_IF
////////////////////////////////////////////////action/////////////////////////////////////////////
		E_WorkingStates.TOTE_LOAD:	
			workflow_status	:= ToteSubsystemWorkflowStatus.INBOUNDING;
			ton_timeout.PT	:= T#5S;	
			roller_inbound.roller.forward	:= TRUE;
			IF roller_inbound.photo_sensor.Q THEN	
				roller_inbound.roller.forward	:= FALSE;
				eStates	:= E_WorkingStates.BAG_OPEN_DOWN;
			END_IF
		E_WorkingStates.BAG_OPEN_DOWN:
			ton_timeout.PT	:= T#5S;
			workflow_status	:= ToteSubsystemWorkflowStatus.BAG_OPENING;
			st_mcAxis_lift.mcMoveAbsolute.Execute	:= TRUE;		
			st_mcAxis_lift.rActualPosSet	:= rPos_lift_down;
			st_mcAxis_lift.rVelocitySet	:= 250;
			IF st_mcAxis_lift.mcMoveAbsolute.Done THEN
				
				eStates	:= E_WorkingStates.VACUUN_ON;
			END_IF		
			
		E_WorkingStates.VACUUN_ON:
			ton_timeout.PT	:=T#10MS;
			valve_vacuun[0].extend	:= TRUE;
			valve_vacuun[1].extend	:= TRUE;
			valve_vacuun[2].extend	:= TRUE;
			valve_vacuun[3].extend	:= TRUE;
//			IF valve_vacuun[0].extended AND valve_vacuun[1].extended AND valve_vacuun[2].extended AND valve_vacuun[3].extended THEN
//				eStates	:= E_WorkingStates.BAG_OPEN_VACUUN_BEGIN;
//			END_IF
			IF ton_timeout.Q THEN
				eStates	:= E_WorkingStates.BAG_OPEN_VACUUN_BEGIN;
			END_IF
		E_WorkingStates.BAG_OPEN_VACUUN_BEGIN:	
			ton_timeout.PT	:=T#5S;		
			st_mcAxis_vacuun[0].mcMoveAbsolute.Execute	:= TRUE;		
			st_mcAxis_vacuun[0].rActualPosSet	:= rPos_vacuun_home[0];
			st_mcAxis_vacuun[0].rVelocitySet	:= 300;
			st_mcAxis_vacuun[1].mcMoveAbsolute.Execute	:= TRUE;		
			st_mcAxis_vacuun[1].rActualPosSet	:= rPos_vacuun_home[1];
			st_mcAxis_vacuun[1].rVelocitySet	:= 300;
			IF st_mcAxis_vacuun[0].mcMoveAbsolute.Done AND st_mcAxis_vacuun[1].mcMoveAbsolute.Done THEN
				st_mcAxis_vacuun[0].mcMoveAbsolute.Execute	:= FALSE;
				st_mcAxis_vacuun[1].mcMoveAbsolute.Execute	:= FALSE;
				eStates	:= E_WorkingStates.WAIT;
			END_IF
		E_WorkingStates.WAIT:
			ton_timeout.PT	:= T#2000MS;
			//roller_inbound.roller.forward	:= TRUE;
			IF ton_timeout.Q OR (valve_vacuun[0].extended AND valve_vacuun[1].extended AND valve_vacuun[2].extended AND valve_vacuun[3].extended) THEN
				tote_status	:= ToteStatus.LOADED;
				//roller_inbound.roller.forward	:= FALSE;
				eStates	:= E_WorkingStates.WAIT_1;
			END_IF
		E_WorkingStates.WAIT_1:
			ton_timeout.PT	:= T#300MS;
			IF ton_timeout.Q THEN
				eStates	:= E_WorkingStates.BAG_OPEN_AXIS_OPEN;
			END_IF
		E_WorkingStates.BAG_OPEN_AXIS_OPEN:
			ton_timeout.PT	:=T#5S;
			st_mcAxis_vacuun[0].mcMoveAbsolute.Execute	:= TRUE;		
			st_mcAxis_vacuun[0].rActualPosSet	:= rPos_vacuun_working[0];
			st_mcAxis_vacuun[0].rVelocitySet	:= 200;
			st_mcAxis_vacuun[1].mcMoveAbsolute.Execute	:= TRUE;		
			st_mcAxis_vacuun[1].rActualPosSet	:= rPos_vacuun_working[1];
			st_mcAxis_vacuun[1].rVelocitySet	:= 200;
			IF st_mcAxis_vacuun[0].mcMoveAbsolute.Done AND st_mcAxis_vacuun[1].mcMoveAbsolute.Done THEN
				st_mcAxis_vacuun[0].mcMoveAbsolute.Execute	:= FALSE;
				st_mcAxis_vacuun[1].mcMoveAbsolute.Execute	:= FALSE;
				eStates	:= E_WorkingStates.BAG_OPEN_AXIS_CYCLINDER_DOWN;
			END_IF		
		E_WorkingStates.BAG_OPEN_AXIS_CYCLINDER_DOWN:
			ton_timeout.PT	:=T#1S;
			valve_open_lift.extend	:= TRUE;
			valve_open_lift.retract	:= FALSE;
			IF valve_open_lift.extended AND NOT valve_open_lift.retracted THEN
				eStates	:= E_WorkingStates.BAG_OPEN;
			END_IF
			IF ton_timeout.Q THEN
				eStates	:= E_WorkingStates.BAG_OPEN;
			END_IF
		E_WorkingStates.BAG_OPEN:
			ton_timeout.PT	:=T#5S;
			valve_open_side.extend	:= TRUE;
			valve_open_side.retract	:= FALSE;
			st_mcAxis_bagOpen[0].mcMoveAbsolute.Execute	:= TRUE;		
			st_mcAxis_bagOpen[0].rActualPosSet	:= rPos_bag_end[0];
			st_mcAxis_bagOpen[0].rVelocitySet	:= 150;			
			st_mcAxis_bagOpen[1].mcMoveAbsolute.Execute	:= TRUE;		
			st_mcAxis_bagOpen[1].rActualPosSet	:= rPos_bag_end[1];
			st_mcAxis_bagOpen[1].rVelocitySet	:= 150;				
			st_mcAxis_bagOpen[2].mcMoveAbsolute.Execute	:= TRUE;		
			st_mcAxis_bagOpen[2].rActualPosSet	:= rPos_bag_end[2];
			st_mcAxis_bagOpen[2].rVelocitySet	:= 150;				
			st_mcAxis_bagOpen[3].mcMoveAbsolute.Execute	:= TRUE;		
			st_mcAxis_bagOpen[3].rActualPosSet	:= rPos_bag_end[3];
			st_mcAxis_bagOpen[3].rVelocitySet	:= 150;				
			IF ((valve_open_side.extended AND NOT valve_open_side.retracted) OR ton_timeout.Q) AND st_mcAxis_bagOpen[0].mcMoveAbsolute.Done 
			AND st_mcAxis_bagOpen[1].mcMoveAbsolute.Done AND st_mcAxis_bagOpen[2].mcMoveAbsolute.Done AND st_mcAxis_bagOpen[3].mcMoveAbsolute.Done THEN	
				eStates	:= E_WorkingStates.VACUUN_OFF;
			END_IF
		E_WorkingStates.VACUUN_OFF:
			ton_timeout.PT	:=T#1S;
			valve_vacuun[0].extend	:= FALSE;
			valve_vacuun[1].extend	:= FALSE;
			valve_vacuun[2].extend	:= FALSE;
			valve_vacuun[3].extend	:= FALSE;
			IF NOT (valve_vacuun[0].extended OR valve_vacuun[1].extended OR valve_vacuun[2].extended OR valve_vacuun[3].extended) THEN
				eStates	:= E_WorkingStates.DONE;
			END_IF
			IF ton_timeout.Q THEN
				eStates	:= E_WorkingStates.DONE;
			END_IF
		E_WorkingStates.DONE:
			ADSLOGSTR(msgCtrlMask:= ADSLOG_MSGTYPE_LOG,msgFmtStr:='load end',strArg:='');
			tote_status	:= ToteStatus.READY;
			workflow_status	:= ToteSubsystemWorkflowStatus.IDLE;	
			M_load	:= TRUE;
			xLoading	:= FALSE;
			eStates	:= E_WorkingStates.IDLE;
		E_WorkingStates.ERROR:
			xError	:=	TRUE;
			workflow_status	:= ToteSubsystemWorkflowStatus.IDLE;
			roller_inbound.roller.forward		:= FALSE;	
			st_mcAxis_vacuun[0].mcMoveAbsolute.Execute	:= FALSE;
			st_mcAxis_vacuun[1].mcMoveAbsolute.Execute	:= FALSE;
			st_mcAxis_bagOpen[0].mcMoveAbsolute.Execute	:= FALSE;
			st_mcAxis_bagOpen[1].mcMoveAbsolute.Execute	:= FALSE;
			st_mcAxis_bagOpen[2].mcMoveAbsolute.Execute	:= FALSE;
			st_mcAxis_bagOpen[3].mcMoveAbsolute.Execute	:= FALSE;
			st_mcAxis_lift.mcMoveAbsolute.Execute	:= FALSE;			
			M_load 		:= TRUE;
		
END_CASE
END_METHOD

METHOD M_mapping : BOOL
VAR_INPUT
END_VAR
event.sTime	:= MAIN.Temp_str;
event.sComponent_name	:= sComponent_name;
/////////////////////////////////////digital input////////////////////////////////////////
valve_lift.extended					:= G_IO.arDI[5].Ch[0] OR G_IO.arDI[5].Ch[2];
valve_lift.retracted				:= G_IO.arDI[5].Ch[1] OR G_IO.arDI[5].Ch[3];
roller_inbound.photo_sensor_mute(D:= G_IO.arDI[5].Ch[4],on_ms:=10,off_ms:=100);
roller_inbound.roller.err			:= G_IO.arDI[5].Ch[5];
roller_inbound.photo_sensor(D:= G_IO.arDI[5].Ch[6],on_ms:=100,off_ms:=100);
roller_outbound.roller.err			:= G_IO.arDI[5].Ch[7];
roller_outbound.photo_sensor(D:= G_IO.arDI[5].Ch[8],on_ms:=100,off_ms:=500);		
sensor_openbag_detection[0]			:= G_IO.arDI[5].Ch[9];
sensor_openbag_detection[1]			:= G_IO.arDI[5].Ch[10];
sensor_openbag_detection[2]			:= G_IO.arDI[5].Ch[11];
sensor_openbag_detection[3]			:= G_IO.arDI[5].Ch[12];
sensor_openbag_detection[4]			:= G_IO.arDI[5].Ch[13];
sensor_openbag_detection[5]			:= G_IO.arDI[5].Ch[14];
sensor_openbag_detection[6]			:= G_IO.arDI[5].Ch[15];
sensor_openbag_detection[7]			:= G_IO.arDI[6].Ch[0];
sensor_cover[0]						:= G_IO.arDI[6].Ch[1];
sensor_cover[1]						:= G_IO.arDI[6].Ch[2];
EDM_KA10							:= G_IO.arDI[6].Ch[3];
roller_outbound_end.roller.err		:= G_IO.arDI[6].Ch[4];

bag_open_detection[0](D:=G_IO.arDI[7].Ch[9],on_ms:=,off_ms:=);
bag_open_detection[0](D:=G_IO.arDI[7].Ch[10],on_ms:=,off_ms:=);
bag_open_detection[0](D:=G_IO.arDI[7].Ch[11],on_ms:=,off_ms:=);
bag_open_detection[0](D:=G_IO.arDI[7].Ch[12],on_ms:=,off_ms:=);

valve_vacuun[0].extended		:= G_IO.arDI[8].Ch[6];
valve_vacuun[1].extended		:= G_IO.arDI[8].Ch[7];
valve_vacuun[2].extended		:= G_IO.arDI[8].Ch[8];
valve_vacuun[3].extended		:= G_IO.arDI[8].Ch[9];
valve_open_side.extended		:= G_IO.arDI[8].Ch[11];
valve_open_side.retracted		:= G_IO.arDI[8].Ch[10];
valve_open_lift.extended		:= G_IO.arDI[8].Ch[12];
valve_open_lift.retracted		:= G_IO.arDI[8].Ch[13];

